LIN {X 0,Y 422.066,Z 378.159,A -85,B 0,C 180,E1 -10186.597,E2 -10186.597} C_VEL
LIN {X 0,Y 422.405,Z 363.356,A -85,B 0,C 180,E1 -10186.926,E2 -10186.926} C_VEL
LIN {X 0,Y 423.125,Z 289.794,A -85,B 0,C 180,E1 -10188.266,E2 -10188.266} C_VEL
LIN {X 0,Y 419.451,Z 264.662,A -85,B 0,C 180,E1 -10188.909,E2 -10188.909} C_VEL
LIN {X 0,Y 420.506,Z 247.774,A -85,B 0,C 180,E1 -10192.086,E2 -10192.086} C_VEL
LIN {X 0,Y 421.39,Z 234.372,A -85,B 0,C 180,E1 -10194.639,E2 -10194.639} C_VEL
LIN {X 0,Y 420.674,Z 228.931,A -85,B 0,C 180,E1 -10195.742,E2 -10195.742} C_VEL
LIN {X 0,Y 418.333,Z 217.378,A -85,B 0,C 180,E1 -10198.193,E2 -10198.193} C_VEL
LIN {X 0,Y 418.2,Z 217.392,A -85,B 0,C 180,E1 -10201.393,E2 -10201.393} C_VEL
LIN {X 0,Y 418.252,Z 217.383,A -85,B 0,C 180,E1 -10204.577,E2 -10204.577} C_VEL
LIN {X 0,Y 418.211,Z 217.393,A -85,B 0,C 180,E1 -10207.83,E2 -10207.83} C_VEL
LIN {X 0,Y 418.203,Z 217.388,A -85,B 0,C 180,E1 -10210.945,E2 -10210.945} C_VEL
LIN {X 0,Y 418.188,Z 217.396,A -85,B 0,C 180,E1 -10213.726,E2 -10213.726} C_VEL
LIN {X 0,Y 418.184,Z 217.391,A -85,B 0,C 180,E1 -10216.445,E2 -10216.445} C_VEL
LIN {X 0,Y 418.196,Z 217.39,A -85,B 0,C 180,E1 -10219.127,E2 -10219.127} C_VEL
LIN {X 0,Y 418.195,Z 217.391,A -85,B 0,C 180,E1 -10222.164,E2 -10222.164} C_VEL
LIN {X 0,Y 418.234,Z 217.389,A -85,B 0,C 180,E1 -10225.417,E2 -10225.417} C_VEL
LIN {X 0,Y 418.176,Z 217.391,A -85,B 0,C 180,E1 -10228.601,E2 -10228.601} C_VEL
LIN {X 0,Y 418.254,Z 217.384,A -85,B 0,C 180,E1 -10231.934,E2 -10231.934} C_VEL
LIN {X 0,Y 418.253,Z 217.386,A -85,B 0,C 180,E1 -10235.16,E2 -10235.16} C_VEL
LIN {X 0,Y 418.192,Z 217.389,A -85,B 0,C 180,E1 -10238.301,E2 -10238.301} C_VEL
LIN {X 0,Y 418.24,Z 217.389,A -85,B 0,C 180,E1 -10241.381,E2 -10241.381} C_VEL
LIN {X 0,Y 418.255,Z 217.381,A -85,B 0,C 180,E1 -10244.404,E2 -10244.404} C_VEL
LIN {X 0,Y 418.324,Z 217.377,A -85,B 0,C 180,E1 -10247.384,E2 -10247.384} C_VEL
LIN {X 0,Y 418.297,Z 217.376,A -85,B 0,C 180,E1 -10250.327,E2 -10250.327} C_VEL
LIN {X 0,Y 418.44,Z 217.363,A -85,B 0,C 180,E1 -10253.248,E2 -10253.248} C_VEL
LIN {X 0,Y 418.287,Z 217.383,A -85,B 0,C 180,E1 -10255.181,E2 -10255.181} C_VEL
LIN {X 0,Y 418.492,Z 217.352,A -85,B 0,C 180,E1 -10258.075,E2 -10258.075} C_VEL
LIN {X 0,Y 418.62,Z 217.336,A -85,B 0,C 180,E1 -10260,E2 -10260} C_VEL
LIN {X 0,Y 418.452,Z 217.364,A -85,B 0,C 180,E1 -10262.888,E2 -10262.888} C_VEL
LIN {X 0,Y 418.491,Z 217.352,A -85,B 0,C 180,E1 -10265.783,E2 -10265.783} C_VEL
LIN {X 0,Y 418.354,Z 217.376,A -85,B 0,C 180,E1 -10268.696,E2 -10268.696} C_VEL
LIN {X 0,Y 418.289,Z 217.377,A -85,B 0,C 180,E1 -10271.631,E2 -10271.631} C_VEL
LIN {X 0,Y 418.264,Z 217.387,A -85,B 0,C 180,E1 -10274.598,E2 -10274.598} C_VEL
LIN {X 0,Y 418.244,Z 217.383,A -85,B 0,C 180,E1 -10277.605,E2 -10277.605} C_VEL
LIN {X 0,Y 418.245,Z 217.388,A -85,B 0,C 180,E1 -10280.663,E2 -10280.663} C_VEL
LIN {X 0,Y 418.263,Z 217.381,A -85,B 0,C 180,E1 -10283.782,E2 -10283.782} C_VEL
LIN {X 0,Y 418.272,Z 217.38,A -85,B 0,C 180,E1 -10287.073,E2 -10287.073} C_VEL
LIN {X 0,Y 418.222,Z 217.392,A -85,B 0,C 180,E1 -10290.274,E2 -10290.274} C_VEL
LIN {X 0,Y 418.213,Z 217.388,A -85,B 0,C 180,E1 -10293.68,E2 -10293.68} C_VEL
LIN {X 0,Y 418.214,Z 217.386,A -85,B 0,C 180,E1 -10297.226,E2 -10297.226} C_VEL
LIN {X 0,Y 418.237,Z 217.385,A -85,B 0,C 180,E1 -10299.683,E2 -10299.683} C_VEL
LIN {X 0,Y 418.256,Z 217.386,A -85,B 0,C 180,E1 -10302.332,E2 -10302.332} C_VEL
LIN {X 0,Y 418.219,Z 217.386,A -85,B 0,C 180,E1 -10305.113,E2 -10305.113} C_VEL
LIN {X 0,Y 418.232,Z 217.388,A -85,B 0,C 180,E1 -10307.772,E2 -10307.772} C_VEL
LIN {X 0,Y 418.245,Z 217.383,A -85,B 0,C 180,E1 -10310.62,E2 -10310.62} C_VEL
LIN {X 0,Y 418.227,Z 217.391,A -85,B 0,C 180,E1 -10313.979,E2 -10313.979} C_VEL
LIN {X 0,Y 418.241,Z 217.384,A -85,B 0,C 180,E1 -10317.159,E2 -10317.159} C_VEL
LIN {X 0,Y 418.261,Z 217.381,A -85,B 0,C 180,E1 -10320.841,E2 -10320.841} C_VEL
LIN {X 0,Y 418.26,Z 217.383,A -85,B 0,C 180,E1 -10324.098,E2 -10324.098} C_VEL
LIN {X 0,Y 418.229,Z 217.387,A -85,B 0,C 180,E1 -10327.266,E2 -10327.266} C_VEL
LIN {X 0,Y 418.276,Z 217.379,A -85,B 0,C 180,E1 -10330.366,E2 -10330.366} C_VEL
LIN {X 0,Y 418.312,Z 217.38,A -85,B 0,C 180,E1 -10333.406,E2 -10333.406} C_VEL
LIN {X 0,Y 418.342,Z 217.373,A -85,B 0,C 180,E1 -10337.001,E2 -10337.001} C_VEL
LIN {X 0,Y 418.339,Z 217.371,A -85,B 0,C 180,E1 -10340.33,E2 -10340.33} C_VEL
LIN {X 0,Y 418.485,Z 217.359,A -85,B 0,C 180,E1 -10343.25,E2 -10343.25} C_VEL
LIN {X 0,Y 418.336,Z 217.377,A -85,B 0,C 180,E1 -10345.182,E2 -10345.182} C_VEL
LIN {X 0,Y 418.542,Z 217.346,A -85,B 0,C 180,E1 -10348.076,E2 -10348.076} C_VEL
LIN {X 0,Y 418.67,Z 217.33,A -85,B 0,C 180,E1 -10350,E2 -10350} C_VEL
LIN {X 0,Y 418.509,Z 217.354,A -85,B 0,C 180,E1 -10352.887,E2 -10352.887} C_VEL
LIN {X 0,Y 418.501,Z 217.351,A -85,B 0,C 180,E1 -10355.782,E2 -10355.782} C_VEL
LIN {X 0,Y 418.394,Z 217.367,A -85,B 0,C 180,E1 -10358.694,E2 -10358.694} C_VEL
LIN {X 0,Y 418.313,Z 217.375,A -85,B 0,C 180,E1 -10361.63,E2 -10361.63} C_VEL
LIN {X 0,Y 418.316,Z 217.376,A -85,B 0,C 180,E1 -10363.378,E2 -10363.378} C_VEL
LIN {X 0,Y 417.625,Z 217.461,A -85,B 0,C 180,E1 -10364.181,E2 -10364.181} C_VEL
LIN {X 0,Y 414.745,Z 217.82,A -85,B 0,C 180,E1 -10365.486,E2 -10365.486} C_VEL
LIN {X 0,Y 412.331,Z 218.122,A -85,B 0,C 180,E1 -10366.54,E2 -10366.54} C_VEL
LIN {X 0,Y 411.31,Z 218.249,A -85,B 0,C 180,E1 -10367.355,E2 -10367.355} C_VEL
LIN {X 0,Y 411.235,Z 218.256,A -85,B 0,C 180,E1 -10367.631,E2 -10367.631} C_VEL
LIN {X 0,Y 411.189,Z 218.266,A -85,B 0,C 180,E1 -10371.032,E2 -10371.032} C_VEL
LIN {X 0,Y 411.211,Z 218.26,A -85,B 0,C 180,E1 -10374.214,E2 -10374.214} C_VEL
LIN {X 0,Y 411.253,Z 218.258,A -85,B 0,C 180,E1 -10377.475,E2 -10377.475} C_VEL
LIN {X 0,Y 411.299,Z 218.345,A -85,B 0,C 180,E1 -10378.511,E2 -10378.511} C_VEL
LIN {X 0,Y 412.921,Z 227.389,A -85,B 0,C 180,E1 -10380.701,E2 -10380.701} C_VEL
LIN {X 0,Y 412.961,Z 228.338,A -85,B 0,C 180,E1 -10380.91,E2 -10380.91} C_VEL
LIN {X 0,Y 416.873,Z 248.303,A -85,B 0,C 180,E1 -10381.469,E2 -10381.469} C_VEL
LIN {X 0,Y 415.524,Z 335.93,A -85,B 0,C 180,E1 -10383.106,E2 -10383.106} C_VEL
LIN {X 0,Y 415.093,Z 349.118,A -85,B 0,C 180,E1 -10383.544,E2 -10383.544} C_VEL
LIN {X 0,Y 414.718,Z 361.357,A -85,B 0,C 180,E1 -10384.145,E2 -10384.145} C_VEL
LIN {X 0,Y 414.124,Z 373.394,A -85,B 0,C 180,E1 -10384.939,E2 -10384.939} C_VEL
LIN {X 0,Y 413.426,Z 384.953,A -85,B 0,C 180,E1 -10385.923,E2 -10385.923} C_VEL
LIN {X 0,Y 412.769,Z 395.514,A -85,B 0,C 180,E1 -10387.049,E2 -10387.049} C_VEL
LIN {X 0,Y 412.088,Z 405.097,A -85,B 0,C 180,E1 -10388.325,E2 -10388.325} C_VEL
LIN {X 0,Y 411.513,Z 413.918,A -85,B 0,C 180,E1 -10389.778,E2 -10389.778} C_VEL
LIN {X 0,Y 410.989,Z 420.898,A -85,B 0,C 180,E1 -10391.201,E2 -10391.201} C_VEL
LIN {X 0,Y 410.643,Z 426.469,A -85,B 0,C 180,E1 -10392.615,E2 -10392.615} C_VEL
LIN {X 0,Y 410.38,Z 430.837,A -85,B 0,C 180,E1 -10394.006,E2 -10394.006} C_VEL
LIN {X 0,Y 410.192,Z 434.163,A -85,B 0,C 180,E1 -10395.375,E2 -10395.375} C_VEL
LIN {X 0,Y 410.001,Z 436.573,A -85,B 0,C 180,E1 -10396.713,E2 -10396.713} C_VEL
LIN {X 0,Y 409.91,Z 438.196,A -85,B 0,C 180,E1 -10398.036,E2 -10398.036} C_VEL
LIN {X 0,Y 409.864,Z 439.072,A -85,B 0,C 180,E1 -10399.339,E2 -10399.339} C_VEL
LIN {X 0,Y 409.87,Z 439.206,A -85,B 0,C 180,E1 -10400.622,E2 -10400.622} C_VEL
LIN {X 0,Y 409.899,Z 438.569,A -85,B 0,C 180,E1 -10402.056,E2 -10402.056} C_VEL
LIN {X 0,Y 410.047,Z 436.829,A -85,B 0,C 180,E1 -10403.655,E2 -10403.655} C_VEL
LIN {X 0,Y 410.286,Z 433.278,A -85,B 0,C 180,E1 -10405.579,E2 -10405.579} C_VEL
LIN {X 0,Y 410.745,Z 427.943,A -85,B 0,C 180,E1 -10407.486,E2 -10407.486} C_VEL
LIN {X 0,Y 411.237,Z 421.689,A -85,B 0,C 180,E1 -10409.157,E2 -10409.157} C_VEL
LIN {X 0,Y 411.863,Z 414.212,A -85,B 0,C 180,E1 -10410.706,E2 -10410.706} C_VEL
LIN {X 0,Y 412.617,Z 405.207,A -85,B 0,C 180,E1 -10412.198,E2 -10412.198} C_VEL
LIN {X 0,Y 413.328,Z 395.464,A -85,B 0,C 180,E1 -10413.491,E2 -10413.491} C_VEL
LIN {X 0,Y 414.031,Z 385.541,A -85,B 0,C 180,E1 -10414.554,E2 -10414.554} C_VEL
LIN {X 0,Y 414.867,Z 374.104,A -85,B 0,C 180,E1 -10415.532,E2 -10415.532} C_VEL
LIN {X 0,Y 415.491,Z 362.385,A -85,B 0,C 180,E1 -10416.314,E2 -10416.314} C_VEL
LIN {X 0,Y 416.081,Z 349.135,A -85,B 0,C 180,E1 -10416.959,E2 -10416.959} C_VEL
LIN {X 0,Y 416.423,Z 336.373,A -85,B 0,C 180,E1 -10417.382,E2 -10417.382} C_VEL
LIN {X 0,Y 417.941,Z 247.923,A -85,B 0,C 180,E1 -10419.072,E2 -10419.072} C_VEL
LIN {X 0,Y 413.701,Z 229.623,A -85,B 0,C 180,E1 -10419.685,E2 -10419.685} C_VEL
LIN {X 0,Y 413.487,Z 228.755,A -85,B 0,C 180,E1 -10419.738,E2 -10419.738} C_VEL
LIN {X 0,Y 411.235,Z 218.26,A -85,B 0,C 180,E1 -10422.085,E2 -10422.085} C_VEL
LIN {X 0,Y 411.222,Z 218.266,A -85,B 0,C 180,E1 -10425.146,E2 -10425.146} C_VEL
LIN {X 0,Y 411.257,Z 218.262,A -85,B 0,C 180,E1 -10428.167,E2 -10428.167} C_VEL
LIN {X 0,Y 411.4,Z 218.239,A -85,B 0,C 180,E1 -10432.185,E2 -10432.185} C_VEL
LIN {X 0,Y 411.448,Z 218.232,A -85,B 0,C 180,E1 -10434.118,E2 -10434.118} C_VEL
LIN {X 0,Y 411.462,Z 218.23,A -85,B 0,C 180,E1 -10438.043,E2 -10438.043} C_VEL
LIN {X 0,Y 411.591,Z 218.214,A -85,B 0,C 180,E1 -10440,E2 -10440} C_VEL
LIN {X 0,Y 411.409,Z 218.239,A -85,B 0,C 180,E1 -10442.938,E2 -10442.938} C_VEL
LIN {X 0,Y 411.406,Z 218.24,A -85,B 0,C 180,E1 -10446.868,E2 -10446.868} C_VEL
LIN {X 0,Y 411.251,Z 218.255,A -85,B 0,C 180,E1 -10449.84,E2 -10449.84} C_VEL
LIN {X 0,Y 411.27,Z 218.255,A -85,B 0,C 180,E1 -10453.109,E2 -10453.109} C_VEL
LIN {X 0,Y 411.22,Z 218.259,A -85,B 0,C 180,E1 -10456.891,E2 -10456.891} C_VEL
LIN {X 0,Y 411.17,Z 218.265,A -85,B 0,C 180,E1 -10459.99,E2 -10459.99} C_VEL
LIN {X 0,Y 411.158,Z 218.264,A -85,B 0,C 180,E1 -10463.151,E2 -10463.151} C_VEL
LIN {X 0,Y 411.202,Z 218.263,A -85,B 0,C 180,E1 -10466.384,E2 -10466.384} C_VEL
LIN {X 0,Y 411.166,Z 218.262,A -85,B 0,C 180,E1 -10469.716,E2 -10469.716} C_VEL
LIN {X 0,Y 411.176,Z 218.264,A -85,B 0,C 180,E1 -10473.159,E2 -10473.159} C_VEL
LIN {X 0,Y 411.163,Z 218.271,A -85,B 0,C 180,E1 -10476.555,E2 -10476.555} C_VEL
LIN {X 0,Y 411.181,Z 218.266,A -85,B 0,C 180,E1 -10479.73,E2 -10479.73} C_VEL
LIN {X 0,Y 411.148,Z 218.265,A -85,B 0,C 180,E1 -10483.137,E2 -10483.137} C_VEL
LIN {X 0,Y 411.147,Z 218.269,A -85,B 0,C 180,E1 -10485.885,E2 -10485.885} C_VEL
LIN {X 0,Y 411.145,Z 218.27,A -85,B 0,C 180,E1 -10488.775,E2 -10488.775} C_VEL
LIN {X 0,Y 411.177,Z 218.268,A -85,B 0,C 180,E1 -10492.029,E2 -10492.029} C_VEL
LIN {X 0,Y 411.193,Z 218.266,A -85,B 0,C 180,E1 -10495.67,E2 -10495.67} C_VEL
LIN {X 0,Y 411.179,Z 218.267,A -85,B 0,C 180,E1 -10499.155,E2 -10499.155} C_VEL
LIN {X 0,Y 411.273,Z 218.415,A -85,B 0,C 180,E1 -10501.627,E2 -10501.627} C_VEL
LIN {X 0,Y 413.841,Z 230.347,A -85,B 0,C 180,E1 -10504.167,E2 -10504.167} C_VEL
LIN {X 0,Y 414.527,Z 235.409,A -85,B 0,C 180,E1 -10505.192,E2 -10505.192} C_VEL
LIN {X 0,Y 413.41,Z 251.975,A -85,B 0,C 180,E1 -10508.302,E2 -10508.302} C_VEL
LIN {X 0,Y 412.777,Z 262.59,A -85,B 0,C 180,E1 -10510.278,E2 -10510.278} C_VEL
LIN {X 0,Y 416.024,Z 282.027,A -85,B 0,C 180,E1 -10510.862,E2 -10510.862} C_VEL
LIN {X 0,Y 417.333,Z 292.66,A -85,B 0,C 180,E1 -10511.141,E2 -10511.141} C_VEL
LIN {X 0,Y 416.124,Z 372.966,A -85,B 0,C 180,E1 -10512.684,E2 -10512.684} C_VEL
LIN {X 0,Y 415.444,Z 386.355,A -85,B 0,C 180,E1 -10513.13,E2 -10513.13} C_VEL
LIN {X 0,Y 414.759,Z 399.136,A -85,B 0,C 180,E1 -10513.766,E2 -10513.766} C_VEL
LIN {X 0,Y 413.911,Z 411.684,A -85,B 0,C 180,E1 -10514.617,E2 -10514.617} C_VEL
LIN {X 0,Y 413.088,Z 423.323,A -85,B 0,C 180,E1 -10515.632,E2 -10515.632} C_VEL
LIN {X 0,Y 412.332,Z 433.101,A -85,B 0,C 180,E1 -10516.698,E2 -10516.698} C_VEL
LIN {X 0,Y 411.651,Z 442.324,A -85,B 0,C 180,E1 -10517.929,E2 -10517.929} C_VEL
LIN {X 0,Y 410.915,Z 451.346,A -85,B 0,C 180,E1 -10519.406,E2 -10519.406} C_VEL
LIN {X 0,Y 410.467,Z 458.597,A -85,B 0,C 180,E1 -10520.888,E2 -10520.888} C_VEL
LIN {X 0,Y 410.176,Z 465.224,A -85,B 0,C 180,E1 -10522.617,E2 -10522.617} C_VEL
LIN {X 0,Y 409.99,Z 469.606,A -85,B 0,C 180,E1 -10524.097,E2 -10524.097} C_VEL
LIN {X 0,Y 410.011,Z 471.94,A -85,B 0,C 180,E1 -10525.084,E2 -10525.084} C_VEL
LIN {X 0,Y 409.941,Z 473.79,A -85,B 0,C 180,E1 -10526.068,E2 -10526.068} C_VEL
LIN {X 0,Y 409.971,Z 475.198,A -85,B 0,C 180,E1 -10527.052,E2 -10527.052} C_VEL
LIN {X 0,Y 410.019,Z 476.203,A -85,B 0,C 180,E1 -10528.036,E2 -10528.036} C_VEL
LIN {X 0,Y 409.981,Z 476.805,A -85,B 0,C 180,E1 -10529.018,E2 -10529.018} C_VEL
LIN {X 0,Y 409.976,Z 476.961,A -85,B 0,C 180,E1 -10530,E2 -10530} C_VEL
LIN {X 0,Y 409.981,Z 476.707,A -85,B 0,C 180,E1 -10530.982,E2 -10530.982} C_VEL
LIN {X 0,Y 410.018,Z 476.057,A -85,B 0,C 180,E1 -10531.964,E2 -10531.964} C_VEL
LIN {X 0,Y 409.972,Z 474.998,A -85,B 0,C 180,E1 -10532.947,E2 -10532.947} C_VEL
LIN {X 0,Y 409.941,Z 473.471,A -85,B 0,C 180,E1 -10533.932,E2 -10533.932} C_VEL
LIN {X 0,Y 410.024,Z 470.372,A -85,B 0,C 180,E1 -10535.409,E2 -10535.409} C_VEL
LIN {X 0,Y 410.163,Z 466.182,A -85,B 0,C 180,E1 -10536.888,E2 -10536.888} C_VEL
LIN {X 0,Y 410.384,Z 459.759,A -85,B 0,C 180,E1 -10538.617,E2 -10538.617} C_VEL
LIN {X 0,Y 410.732,Z 452.748,A -85,B 0,C 180,E1 -10540.1,E2 -10540.1} C_VEL
LIN {X 0,Y 411.32,Z 443.951,A -85,B 0,C 180,E1 -10541.58,E2 -10541.58} C_VEL
LIN {X 0,Y 411.92,Z 434.928,A -85,B 0,C 180,E1 -10542.813,E2 -10542.813} C_VEL
LIN {X 0,Y 412.682,Z 424.044,A -85,B 0,C 180,E1 -10544.018,E2 -10544.018} C_VEL
LIN {X 0,Y 413.345,Z 412.491,A -85,B 0,C 180,E1 -10545.026,E2 -10545.026} C_VEL
LIN {X 0,Y 414.169,Z 399.868,A -85,B 0,C 180,E1 -10545.878,E2 -10545.878} C_VEL
LIN {X 0,Y 414.792,Z 387.64,A -85,B 0,C 180,E1 -10546.485,E2 -10546.485} C_VEL
LIN {X 0,Y 415.304,Z 374.278,A -85,B 0,C 180,E1 -10546.939,E2 -10546.939} C_VEL
LIN {X 0,Y 415.985,Z 331.19,A -85,B 0,C 180,E1 -10547.758,E2 -10547.758} C_VEL
LIN {X 0,Y 416.299,Z 290.521,A -85,B 0,C 180,E1 -10548.523,E2 -10548.523} C_VEL
LIN {X 0,Y 412.517,Z 264.36,A -85,B 0,C 180,E1 -10549.207,E2 -10549.207} C_VEL
LIN {X 0,Y 413.63,Z 247.327,A -85,B 0,C 180,E1 -10552.473,E2 -10552.473} C_VEL
LIN {X 0,Y 414.434,Z 235.243,A -85,B 0,C 180,E1 -10554.813,E2 -10554.813} C_VEL
LIN {X 0,Y 413.608,Z 229.802,A -85,B 0,C 180,E1 -10555.941,E2 -10555.941} C_VEL
LIN {X 0,Y 411.291,Z 218.254,A -85,B 0,C 180,E1 -10558.442,E2 -10558.442} C_VEL
LIN {X 0,Y 411.154,Z 218.273,A -85,B 0,C 180,E1 -10561.994,E2 -10561.994} C_VEL
LIN {X 0,Y 411.197,Z 218.261,A -85,B 0,C 180,E1 -10564.875,E2 -10564.875} C_VEL
LIN {X 0,Y 411.186,Z 218.266,A -85,B 0,C 180,E1 -10568.165,E2 -10568.165} C_VEL
LIN {X 0,Y 411.144,Z 218.268,A -85,B 0,C 180,E1 -10571.225,E2 -10571.225} C_VEL
LIN {X 0,Y 411.154,Z 218.267,A -85,B 0,C 180,E1 -10574.487,E2 -10574.487} C_VEL
LIN {X 0,Y 411.151,Z 218.268,A -85,B 0,C 180,E1 -10578.191,E2 -10578.191} C_VEL
LIN {X 0,Y 411.18,Z 218.263,A -85,B 0,C 180,E1 -10580.771,E2 -10580.771} C_VEL
LIN {X 0,Y 411.167,Z 218.264,A -85,B 0,C 180,E1 -10584.468,E2 -10584.468} C_VEL
LIN {X 0,Y 411.176,Z 218.264,A -85,B 0,C 180,E1 -10586.87,E2 -10586.87} C_VEL
LIN {X 0,Y 411.18,Z 218.263,A -85,B 0,C 180,E1 -10590.646,E2 -10590.646} C_VEL
LIN {X 0,Y 411.2,Z 218.265,A -85,B 0,C 180,E1 -10593.616,E2 -10593.616} C_VEL
LIN {X 0,Y 411.157,Z 218.267,A -85,B 0,C 180,E1 -10596.849,E2 -10596.849} C_VEL
LIN {X 0,Y 411.172,Z 218.264,A -85,B 0,C 180,E1 -10600.049,E2 -10600.049} C_VEL
LIN {X 0,Y 411.222,Z 218.263,A -85,B 0,C 180,E1 -10603.129,E2 -10603.129} C_VEL
LIN {X 0,Y 411.269,Z 218.255,A -85,B 0,C 180,E1 -10606.891,E2 -10606.891} C_VEL
LIN {X 0,Y 411.25,Z 218.254,A -85,B 0,C 180,E1 -10610.16,E2 -10610.16} C_VEL
LIN {X 0,Y 411.405,Z 218.241,A -85,B 0,C 180,E1 -10613.132,E2 -10613.132} C_VEL
LIN {X 0,Y 411.259,Z 218.259,A -85,B 0,C 180,E1 -10615.098,E2 -10615.098} C_VEL
LIN {X 0,Y 411.461,Z 218.228,A -85,B 0,C 180,E1 -10618.042,E2 -10618.042} C_VEL
LIN {X 0,Y 411.59,Z 218.212,A -85,B 0,C 180,E1 -10620,E2 -10620} C_VEL
LIN {X 0,Y 411.41,Z 218.241,A -85,B 0,C 180,E1 -10622.937,E2 -10622.937} C_VEL
LIN {X 0,Y 411.427,Z 218.237,A -85,B 0,C 180,E1 -10626.762,E2 -10626.762} C_VEL
LIN {X 0,Y 411.251,Z 218.254,A -85,B 0,C 180,E1 -10629.839,E2 -10629.839} C_VEL
LIN {X 0,Y 411.269,Z 218.254,A -85,B 0,C 180,E1 -10633.109,E2 -10633.109} C_VEL
LIN {X 0,Y 411.218,Z 218.262,A -85,B 0,C 180,E1 -10636.89,E2 -10636.89} C_VEL
LIN {X 0,Y 411.216,Z 218.26,A -85,B 0,C 180,E1 -10639.987,E2 -10639.987} C_VEL
LIN {X 0,Y 411.203,Z 218.261,A -85,B 0,C 180,E1 -10643.147,E2 -10643.147} C_VEL
LIN {X 0,Y 411.2,Z 218.267,A -85,B 0,C 180,E1 -10646.383,E2 -10646.383} C_VEL
LIN {X 0,Y 411.172,Z 218.264,A -85,B 0,C 180,E1 -10649.715,E2 -10649.715} C_VEL
LIN {X 0,Y 411.172,Z 218.264,A -85,B 0,C 180,E1 -10653.158,E2 -10653.158} C_VEL
LIN {X 0,Y 411.163,Z 218.268,A -85,B 0,C 180,E1 -10656.556,E2 -10656.556} C_VEL
LIN {X 0,Y 411.199,Z 218.263,A -85,B 0,C 180,E1 -10659.733,E2 -10659.733} C_VEL
LIN {X 0,Y 411.191,Z 218.261,A -85,B 0,C 180,E1 -10663.131,E2 -10663.131} C_VEL
LIN {X 0,Y 411.145,Z 218.272,A -85,B 0,C 180,E1 -10665.884,E2 -10665.884} C_VEL
LIN {X 0,Y 411.189,Z 218.263,A -85,B 0,C 180,E1 -10669.502,E2 -10669.502} C_VEL
LIN {X 0,Y 411.183,Z 218.268,A -85,B 0,C 180,E1 -10672.03,E2 -10672.03} C_VEL
LIN {X 0,Y 411.189,Z 218.266,A -85,B 0,C 180,E1 -10675.669,E2 -10675.669} C_VEL
LIN {X 0,Y 411.183,Z 218.263,A -85,B 0,C 180,E1 -10679.156,E2 -10679.156} C_VEL
LIN {X 0,Y 411.248,Z 218.254,A -85,B 0,C 180,E1 -10682.525,E2 -10682.525} C_VEL
LIN {X 0,Y 411.218,Z 218.264,A -85,B 0,C 180,E1 -10685.787,E2 -10685.787} C_VEL
LIN {X 0,Y 411.188,Z 218.263,A -85,B 0,C 180,E1 -10688.968,E2 -10688.968} C_VEL
LIN {X 0,Y 411.246,Z 218.256,A -85,B 0,C 180,E1 -10692.087,E2 -10692.087} C_VEL
LIN {X 0,Y 411.256,Z 218.256,A -85,B 0,C 180,E1 -10695.149,E2 -10695.149} C_VEL
LIN {X 0,Y 411.281,Z 218.251,A -85,B 0,C 180,E1 -10698.169,E2 -10698.169} C_VEL
LIN {X 0,Y 411.438,Z 218.231,A -85,B 0,C 180,E1 -10702.19,E2 -10702.19} C_VEL
LIN {X 0,Y 411.469,Z 218.227,A -85,B 0,C 180,E1 -10704.119,E2 -10704.119} C_VEL
LIN {X 0,Y 411.512,Z 218.222,A -85,B 0,C 180,E1 -10708.043,E2 -10708.043} C_VEL
LIN {X 0,Y 411.639,Z 218.206,A -85,B 0,C 180,E1 -10710,E2 -10710} C_VEL
LIN {X 0,Y 411.464,Z 218.232,A -85,B 0,C 180,E1 -10712.937,E2 -10712.937} C_VEL
LIN {X 0,Y 411.462,Z 218.228,A -85,B 0,C 180,E1 -10715.882,E2 -10715.882} C_VEL
LIN {X 0,Y 411.349,Z 218.246,A -85,B 0,C 180,E1 -10718.844,E2 -10718.844} C_VEL
LIN {X 0,Y 411.281,Z 218.25,A -85,B 0,C 180,E1 -10721.832,E2 -10721.832} C_VEL
LIN {X 0,Y 411.255,Z 218.26,A -85,B 0,C 180,E1 -10724.851,E2 -10724.851} C_VEL
LIN {X 0,Y 411.235,Z 218.256,A -85,B 0,C 180,E1 -10727.631,E2 -10727.631} C_VEL
LIN {X 0,Y 410.577,Z 218.342,A -85,B 0,C 180,E1 -10728.449,E2 -10728.449} C_VEL
LIN {X 0,Y 407.687,Z 218.698,A -85,B 0,C 180,E1 -10729.777,E2 -10729.777} C_VEL
LIN {X 0,Y 405.239,Z 219.009,A -85,B 0,C 180,E1 -10730.849,E2 -10730.849} C_VEL
LIN {X 0,Y 404.203,Z 219.132,A -85,B 0,C 180,E1 -10731.679,E2 -10731.679} C_VEL
LIN {X 0,Y 404.128,Z 219.141,A -85,B 0,C 180,E1 -10731.961,E2 -10731.961} C_VEL
LIN {X 0,Y 404.206,Z 219.136,A -85,B 0,C 180,E1 -10735.294,E2 -10735.294} C_VEL
LIN {X 0,Y 404.272,Z 219.247,A -85,B 0,C 180,E1 -10738.308,E2 -10738.308} C_VEL
LIN {X 0,Y 405.958,Z 228.546,A -85,B 0,C 180,E1 -10740.599,E2 -10740.599} C_VEL
LIN {X 0,Y 410.088,Z 248.762,A -85,B 0,C 180,E1 -10741.187,E2 -10741.187} C_VEL
LIN {X 0,Y 408.677,Z 336.018,A -85,B 0,C 180,E1 -10742.846,E2 -10742.846} C_VEL
LIN {X 0,Y 408.239,Z 349.273,A -85,B 0,C 180,E1 -10743.292,E2 -10743.292} C_VEL
LIN {X 0,Y 407.832,Z 361.592,A -85,B 0,C 180,E1 -10743.904,E2 -10743.904} C_VEL
LIN {X 0,Y 407.211,Z 373.686,A -85,B 0,C 180,E1 -10744.714,E2 -10744.714} C_VEL
LIN {X 0,Y 406.541,Z 384.676,A -85,B 0,C 180,E1 -10745.659,E2 -10745.659} C_VEL
LIN {X 0,Y 405.838,Z 395.27,A -85,B 0,C 180,E1 -10746.795,E2 -10746.795} C_VEL
LIN {X 0,Y 405.118,Z 405.412,A -85,B 0,C 180,E1 -10748.159,E2 -10748.159} C_VEL
LIN {X 0,Y 404.483,Z 414.468,A -85,B 0,C 180,E1 -10749.678,E2 -10749.678} C_VEL
LIN {X 0,Y 403.967,Z 421.065,A -85,B 0,C 180,E1 -10751.048,E2 -10751.048} C_VEL
LIN {X 0,Y 403.592,Z 426.547,A -85,B 0,C 180,E1 -10752.451,E2 -10752.451} C_VEL
LIN {X 0,Y 403.278,Z 431.818,A -85,B 0,C 180,E1 -10754.188,E2 -10754.188} C_VEL
LIN {X 0,Y 403.041,Z 435.368,A -85,B 0,C 180,E1 -10755.774,E2 -10755.774} C_VEL
LIN {X 0,Y 402.878,Z 437.538,A -85,B 0,C 180,E1 -10757.131,E2 -10757.131} C_VEL
LIN {X 0,Y 402.81,Z 439.001,A -85,B 0,C 180,E1 -10758.604,E2 -10758.604} C_VEL
LIN {X 0,Y 402.754,Z 439.581,A -85,B 0,C 180,E1 -10760.149,E2 -10760.149} C_VEL
LIN {X 0,Y 402.792,Z 439.176,A -85,B 0,C 180,E1 -10761.728,E2 -10761.728} C_VEL
LIN {X 0,Y 402.958,Z 437.329,A -85,B 0,C 180,E1 -10763.631,E2 -10763.631} C_VEL
LIN {X 0,Y 403.215,Z 433.917,A -85,B 0,C 180,E1 -10765.561,E2 -10765.561} C_VEL
LIN {X 0,Y 403.627,Z 429.286,A -85,B 0,C 180,E1 -10767.332,E2 -10767.332} C_VEL
LIN {X 0,Y 404.171,Z 422.865,A -85,B 0,C 180,E1 -10769.139,E2 -10769.139} C_VEL
LIN {X 0,Y 404.745,Z 416.268,A -85,B 0,C 180,E1 -10770.595,E2 -10770.595} C_VEL
LIN {X 0,Y 405.54,Z 407.726,A -85,B 0,C 180,E1 -10772.102,E2 -10772.102} C_VEL
LIN {X 0,Y 406.336,Z 398.021,A -85,B 0,C 180,E1 -10773.476,E2 -10773.476} C_VEL
LIN {X 0,Y 407.023,Z 388.568,A -85,B 0,C 180,E1 -10774.564,E2 -10774.564} C_VEL
LIN {X 0,Y 407.875,Z 377.625,A -85,B 0,C 180,E1 -10775.573,E2 -10775.573} C_VEL
LIN {X 0,Y 408.62,Z 365.339,A -85,B 0,C 180,E1 -10776.458,E2 -10776.458} C_VEL
LIN {X 0,Y 409.269,Z 352.687,A -85,B 0,C 180,E1 -10777.138,E2 -10777.138} C_VEL
LIN {X 0,Y 409.633,Z 339.747,A -85,B 0,C 180,E1 -10777.619,E2 -10777.619} C_VEL
LIN {X 0,Y 410.038,Z 318.579,A -85,B 0,C 180,E1 -10778.07,E2 -10778.07} C_VEL
LIN {X 0,Y 411.313,Z 248.954,A -85,B 0,C 180,E1 -10779.422,E2 -10779.422} C_VEL
LIN {X 0,Y 407.532,Z 232.418,A -85,B 0,C 180,E1 -10779.989,E2 -10779.989} C_VEL
LIN {X 0,Y 406.355,Z 229.099,A -85,B 0,C 180,E1 -10780.159,E2 -10780.159} C_VEL
LIN {X 0,Y 404.185,Z 219.138,A -85,B 0,C 180,E1 -10782.481,E2 -10782.481} C_VEL
LIN {X 0,Y 404.175,Z 219.145,A -85,B 0,C 180,E1 -10785.911,E2 -10785.911} C_VEL
LIN {X 0,Y 404.22,Z 219.14,A -85,B 0,C 180,E1 -10788.975,E2 -10788.975} C_VEL
LIN {X 0,Y 404.363,Z 219.116,A -85,B 0,C 180,E1 -10792.127,E2 -10792.127} C_VEL
LIN {X 0,Y 404.394,Z 219.111,A -85,B 0,C 180,E1 -10794.015,E2 -10794.015} C_VEL
LIN {X 0,Y 404.432,Z 219.106,A -85,B 0,C 180,E1 -10798.009,E2 -10798.009} C_VEL
LIN {X 0,Y 404.561,Z 219.09,A -85,B 0,C 180,E1 -10800,E2 -10800} C_VEL
LIN {X 0,Y 404.367,Z 219.116,A -85,B 0,C 180,E1 -10802.989,E2 -10802.989} C_VEL
LIN {X 0,Y 404.37,Z 219.11,A -85,B 0,C 180,E1 -10805.986,E2 -10805.986} C_VEL
LIN {X 0,Y 404.247,Z 219.13,A -85,B 0,C 180,E1 -10809.002,E2 -10809.002} C_VEL
LIN {X 0,Y 404.225,Z 219.129,A -85,B 0,C 180,E1 -10812.043,E2 -10812.043} C_VEL
LIN {X 0,Y 404.167,Z 219.141,A -85,B 0,C 180,E1 -10815.12,E2 -10815.12} C_VEL
LIN {X 0,Y 404.169,Z 219.137,A -85,B 0,C 180,E1 -10818.24,E2 -10818.24} C_VEL
LIN {X 0,Y 404.098,Z 219.147,A -85,B 0,C 180,E1 -10821.422,E2 -10821.422} C_VEL
LIN {X 0,Y 404.138,Z 219.145,A -85,B 0,C 180,E1 -10824.669,E2 -10824.669} C_VEL
LIN {X 0,Y 404.16,Z 219.139,A -85,B 0,C 180,E1 -10828.003,E2 -10828.003} C_VEL
LIN {X 0,Y 404.106,Z 219.145,A -85,B 0,C 180,E1 -10831.56,E2 -10831.56} C_VEL
LIN {X 0,Y 404.154,Z 219.137,A -85,B 0,C 180,E1 -10835.02,E2 -10835.02} C_VEL
LIN {X 0,Y 404.121,Z 219.147,A -85,B 0,C 180,E1 -10838.761,E2 -10838.761} C_VEL
LIN {X 0,Y 404.096,Z 219.147,A -85,B 0,C 180,E1 -10841.602,E2 -10841.602} C_VEL
LIN {X 0,Y 404.123,Z 219.145,A -85,B 0,C 180,E1 -10844.525,E2 -10844.525} C_VEL
LIN {X 0,Y 404.116,Z 219.144,A -85,B 0,C 180,E1 -10847.299,E2 -10847.299} C_VEL
LIN {X 0,Y 404.153,Z 219.142,A -85,B 0,C 180,E1 -10849.959,E2 -10849.959} C_VEL
LIN {X 0,Y 404.121,Z 219.145,A -85,B 0,C 180,E1 -10853.129,E2 -10853.129} C_VEL
LIN {X 0,Y 404.133,Z 219.146,A -85,B 0,C 180,E1 -10856.191,E2 -10856.191} C_VEL
LIN {X 0,Y 404.136,Z 219.147,A -85,B 0,C 180,E1 -10859.718,E2 -10859.718} C_VEL
LIN {X 0,Y 404.206,Z 219.204,A -85,B 0,C 180,E1 -10861.262,E2 -10861.262} C_VEL
LIN {X 0,Y 406.875,Z 231.415,A -85,B 0,C 180,E1 -10863.923,E2 -10863.923} C_VEL
LIN {X 0,Y 407.635,Z 236.681,A -85,B 0,C 180,E1 -10865.017,E2 -10865.017} C_VEL
LIN {X 0,Y 406.675,Z 250.473,A -85,B 0,C 180,E1 -10867.657,E2 -10867.657} C_VEL
LIN {X 0,Y 405.923,Z 262.373,A -85,B 0,C 180,E1 -10869.893,E2 -10869.893} C_VEL
LIN {X 0,Y 409.282,Z 281.914,A -85,B 0,C 180,E1 -10870.491,E2 -10870.491} C_VEL
LIN {X 0,Y 410.689,Z 294.318,A -85,B 0,C 180,E1 -10870.825,E2 -10870.825} C_VEL
LIN {X 0,Y 409.434,Z 372.565,A -85,B 0,C 180,E1 -10872.36,E2 -10872.36} C_VEL
LIN {X 0,Y 408.679,Z 386.7,A -85,B 0,C 180,E1 -10872.842,E2 -10872.842} C_VEL
LIN {X 0,Y 407.962,Z 399.241,A -85,B 0,C 180,E1 -10873.488,E2 -10873.488} C_VEL
LIN {X 0,Y 407.05,Z 411.699,A -85,B 0,C 180,E1 -10874.351,E2 -10874.351} C_VEL
LIN {X 0,Y 406.21,Z 422.891,A -85,B 0,C 180,E1 -10875.345,E2 -10875.345} C_VEL
LIN {X 0,Y 405.383,Z 433.348,A -85,B 0,C 180,E1 -10876.513,E2 -10876.513} C_VEL
LIN {X 0,Y 404.693,Z 442.162,A -85,B 0,C 180,E1 -10877.719,E2 -10877.719} C_VEL
LIN {X 0,Y 403.903,Z 451.142,A -85,B 0,C 180,E1 -10879.22,E2 -10879.22} C_VEL
LIN {X 0,Y 403.433,Z 458.35,A -85,B 0,C 180,E1 -10880.728,E2 -10880.728} C_VEL
LIN {X 0,Y 403.106,Z 464.961,A -85,B 0,C 180,E1 -10882.487,E2 -10882.487} C_VEL
LIN {X 0,Y 402.919,Z 469.331,A -85,B 0,C 180,E1 -10883.993,E2 -10883.993} C_VEL
LIN {X 0,Y 402.919,Z 471.658,A -85,B 0,C 180,E1 -10884.997,E2 -10884.997} C_VEL
LIN {X 0,Y 402.86,Z 473.493,A -85,B 0,C 180,E1 -10885.999,E2 -10885.999} C_VEL
LIN {X 0,Y 402.947,Z 475.895,A -85,B 0,C 180,E1 -10888.001,E2 -10888.001} C_VEL
LIN {X 0,Y 402.906,Z 476.485,A -85,B 0,C 180,E1 -10889.001,E2 -10889.001} C_VEL
LIN {X 0,Y 402.899,Z 476.627,A -85,B 0,C 180,E1 -10890,E2 -10890} C_VEL
LIN {X 0,Y 402.905,Z 476.364,A -85,B 0,C 180,E1 -10890.999,E2 -10890.999} C_VEL
LIN {X 0,Y 402.946,Z 475.705,A -85,B 0,C 180,E1 -10891.999,E2 -10891.999} C_VEL
LIN {X 0,Y 402.873,Z 474.628,A -85,B 0,C 180,E1 -10892.999,E2 -10892.999} C_VEL
LIN {X 0,Y 402.862,Z 473.085,A -85,B 0,C 180,E1 -10894.001,E2 -10894.001} C_VEL
LIN {X 0,Y 402.921,Z 469.959,A -85,B 0,C 180,E1 -10895.504,E2 -10895.504} C_VEL
LIN {X 0,Y 403.074,Z 465.742,A -85,B 0,C 180,E1 -10897.01,E2 -10897.01} C_VEL
LIN {X 0,Y 403.335,Z 459.287,A -85,B 0,C 180,E1 -10898.769,E2 -10898.769} C_VEL
LIN {X 0,Y 403.685,Z 452.233,A -85,B 0,C 180,E1 -10900.278,E2 -10900.278} C_VEL
LIN {X 0,Y 404.326,Z 443.381,A -85,B 0,C 180,E1 -10901.784,E2 -10901.784} C_VEL
LIN {X 0,Y 404.977,Z 434.306,A -85,B 0,C 180,E1 -10903.037,E2 -10903.037} C_VEL
LIN {X 0,Y 405.689,Z 424.33,A -85,B 0,C 180,E1 -10904.162,E2 -10904.162} C_VEL
LIN {X 0,Y 406.344,Z 413.266,A -85,B 0,C 180,E1 -10905.163,E2 -10905.163} C_VEL
LIN {X 0,Y 407.165,Z 400.918,A -85,B 0,C 180,E1 -10906.03,E2 -10906.03} C_VEL
LIN {X 0,Y 407.831,Z 389.291,A -85,B 0,C 180,E1 -10906.646,E2 -10906.646} C_VEL
LIN {X 0,Y 408.352,Z 377.028,A -85,B 0,C 180,E1 -10907.107,E2 -10907.107} C_VEL
LIN {X 0,Y 408.75,Z 360.306,A -85,B 0,C 180,E1 -10907.477,E2 -10907.477} C_VEL
LIN {X 0,Y 409.571,Z 291.834,A -85,B 0,C 180,E1 -10908.773,E2 -10908.773} C_VEL
LIN {X 0,Y 405.571,Z 264.062,A -85,B 0,C 180,E1 -10909.517,E2 -10909.517} C_VEL
LIN {X 0,Y 406.759,Z 246.836,A -85,B 0,C 180,E1 -10912.874,E2 -10912.874} C_VEL
LIN {X 0,Y 407.471,Z 236.105,A -85,B 0,C 180,E1 -10914.994,E2 -10914.994} C_VEL
LIN {X 0,Y 406.031,Z 227.898,A -85,B 0,C 180,E1 -10916.743,E2 -10916.743} C_VEL
LIN {X 0,Y 404.244,Z 219.132,A -85,B 0,C 180,E1 -10918.7,E2 -10918.7} C_VEL
LIN {X 0,Y 404.129,Z 219.144,A -85,B 0,C 180,E1 -10922.619,E2 -10922.619} C_VEL
LIN {X 0,Y 404.167,Z 219.137,A -85,B 0,C 180,E1 -10925.186,E2 -10925.186} C_VEL
LIN {X 0,Y 404.136,Z 219.14,A -85,B 0,C 180,E1 -10928.754,E2 -10928.754} C_VEL
LIN {X 0,Y 404.103,Z 219.148,A -85,B 0,C 180,E1 -10931.596,E2 -10931.596} C_VEL
LIN {X 0,Y 404.123,Z 219.142,A -85,B 0,C 180,E1 -10934.518,E2 -10934.518} C_VEL
LIN {X 0,Y 404.111,Z 219.145,A -85,B 0,C 180,E1 -10937.292,E2 -10937.292} C_VEL
LIN {X 0,Y 404.129,Z 219.145,A -85,B 0,C 180,E1 -10939.95,E2 -10939.95} C_VEL
LIN {X 0,Y 404.106,Z 219.146,A -85,B 0,C 180,E1 -10943.122,E2 -10943.122} C_VEL
LIN {X 0,Y 404.114,Z 219.144,A -85,B 0,C 180,E1 -10946.184,E2 -10946.184} C_VEL
LIN {X 0,Y 404.111,Z 219.148,A -85,B 0,C 180,E1 -10949.712,E2 -10949.712} C_VEL
LIN {X 0,Y 404.159,Z 219.141,A -85,B 0,C 180,E1 -10953.12,E2 -10953.12} C_VEL
LIN {X 0,Y 404.137,Z 219.146,A -85,B 0,C 180,E1 -10955.331,E2 -10955.331} C_VEL
LIN {X 0,Y 404.097,Z 219.145,A -85,B 0,C 180,E1 -10958.578,E2 -10958.578} C_VEL
LIN {X 0,Y 404.167,Z 219.138,A -85,B 0,C 180,E1 -10961.76,E2 -10961.76} C_VEL
LIN {X 0,Y 404.161,Z 219.14,A -85,B 0,C 180,E1 -10964.88,E2 -10964.88} C_VEL
LIN {X 0,Y 404.224,Z 219.129,A -85,B 0,C 180,E1 -10967.957,E2 -10967.957} C_VEL
LIN {X 0,Y 404.357,Z 219.113,A -85,B 0,C 180,E1 -10972.132,E2 -10972.132} C_VEL
LIN {X 0,Y 404.369,Z 219.111,A -85,B 0,C 180,E1 -10974.014,E2 -10974.014} C_VEL
LIN {X 0,Y 404.43,Z 219.103,A -85,B 0,C 180,E1 -10978.008,E2 -10978.008} C_VEL
LIN {X 0,Y 404.56,Z 219.087,A -85,B 0,C 180,E1 -10980,E2 -10980} C_VEL
LIN {X 0,Y 404.368,Z 219.117,A -85,B 0,C 180,E1 -10982.988,E2 -10982.988} C_VEL
LIN {X 0,Y 404.369,Z 219.114,A -85,B 0,C 180,E1 -10986.764,E2 -10986.764} C_VEL
LIN {X 0,Y 404.217,Z 219.13,A -85,B 0,C 180,E1 -10990.012,E2 -10990.012} C_VEL
LIN {X 0,Y 404.223,Z 219.131,A -85,B 0,C 180,E1 -10993.212,E2 -10993.212} C_VEL
LIN {X 0,Y 404.175,Z 219.138,A -85,B 0,C 180,E1 -10997.009,E2 -10997.009} C_VEL
LIN {X 0,Y 404.17,Z 219.141,A -85,B 0,C 180,E1 -11000.351,E2 -11000.351} C_VEL
LIN {X 0,Y 404.153,Z 219.138,A -85,B 0,C 180,E1 -11003.575,E2 -11003.575} C_VEL
LIN {X 0,Y 404.158,Z 219.139,A -85,B 0,C 180,E1 -11006.879,E2 -11006.879} C_VEL
LIN {X 0,Y 404.116,Z 219.149,A -85,B 0,C 180,E1 -11010.287,E2 -11010.287} C_VEL
LIN {X 0,Y 404.111,Z 219.145,A -85,B 0,C 180,E1 -11013.815,E2 -11013.815} C_VEL
LIN {X 0,Y 404.108,Z 219.144,A -85,B 0,C 180,E1 -11016.878,E2 -11016.878} C_VEL
LIN {X 0,Y 404.139,Z 219.146,A -85,B 0,C 180,E1 -11020.086,E2 -11020.086} C_VEL
LIN {X 0,Y 404.167,Z 219.136,A -85,B 0,C 180,E1 -11023.093,E2 -11023.093} C_VEL
LIN {X 0,Y 404.125,Z 219.147,A -85,B 0,C 180,E1 -11025.929,E2 -11025.929} C_VEL
LIN {X 0,Y 404.128,Z 219.142,A -85,B 0,C 180,E1 -11028.642,E2 -11028.642} C_VEL
LIN {X 0,Y 404.14,Z 219.142,A -85,B 0,C 180,E1 -11031.494,E2 -11031.494} C_VEL
LIN {X 0,Y 404.167,Z 219.136,A -85,B 0,C 180,E1 -11034.987,E2 -11034.987} C_VEL
LIN {X 0,Y 404.13,Z 219.141,A -85,B 0,C 180,E1 -11038.557,E2 -11038.557} C_VEL
LIN {X 0,Y 404.186,Z 219.138,A -85,B 0,C 180,E1 -11042.003,E2 -11042.003} C_VEL
LIN {X 0,Y 404.168,Z 219.139,A -85,B 0,C 180,E1 -11045.337,E2 -11045.337} C_VEL
LIN {X 0,Y 404.13,Z 219.141,A -85,B 0,C 180,E1 -11048.583,E2 -11048.583} C_VEL
LIN {X 0,Y 404.204,Z 219.136,A -85,B 0,C 180,E1 -11051.764,E2 -11051.764} C_VEL
LIN {X 0,Y 404.202,Z 219.133,A -85,B 0,C 180,E1 -11054.884,E2 -11054.884} C_VEL
LIN {X 0,Y 404.253,Z 219.127,A -85,B 0,C 180,E1 -11057.96,E2 -11057.96} C_VEL
LIN {X 0,Y 404.402,Z 219.107,A -85,B 0,C 180,E1 -11062.13,E2 -11062.13} C_VEL
LIN {X 0,Y 404.417,Z 219.106,A -85,B 0,C 180,E1 -11064.016,E2 -11064.016} C_VEL
LIN {X 0,Y 404.481,Z 219.098,A -85,B 0,C 180,E1 -11068.009,E2 -11068.009} C_VEL
LIN {X 0,Y 404.608,Z 219.082,A -85,B 0,C 180,E1 -11070,E2 -11070} C_VEL
LIN {X 0,Y 404.421,Z 219.11,A -85,B 0,C 180,E1 -11072.988,E2 -11072.988} C_VEL
LIN {X 0,Y 404.409,Z 219.106,A -85,B 0,C 180,E1 -11075.985,E2 -11075.985} C_VEL
LIN {X 0,Y 404.287,Z 219.128,A -85,B 0,C 180,E1 -11079,E2 -11079} C_VEL
LIN {X 0,Y 404.253,Z 219.126,A -85,B 0,C 180,E1 -11082.04,E2 -11082.04} C_VEL
LIN {X 0,Y 404.201,Z 219.137,A -85,B 0,C 180,E1 -11085.117,E2 -11085.117} C_VEL
LIN {X 0,Y 404.205,Z 219.133,A -85,B 0,C 180,E1 -11088.236,E2 -11088.236} C_VEL
LIN {X 0,Y 404.131,Z 219.142,A -85,B 0,C 180,E1 -11091.417,E2 -11091.417} C_VEL
LIN {X 0,Y 404.128,Z 219.141,A -85,B 0,C 180,E1 -11091.961,E2 -11091.961} C_VEL
LIN {X 0,Y 403.487,Z 219.228,A -85,B 0,C 180,E1 -11092.792,E2 -11092.792} C_VEL
LIN {X 0,Y 400.653,Z 219.583,A -85,B 0,C 180,E1 -11094.144,E2 -11094.144} C_VEL
LIN {X 0,Y 398.242,Z 219.883,A -85,B 0,C 180,E1 -11095.236,E2 -11095.236} C_VEL
LIN {X 0,Y 397.207,Z 220.009,A -85,B 0,C 180,E1 -11096.081,E2 -11096.081} C_VEL
LIN {X 0,Y 397.124,Z 220.018,A -85,B 0,C 180,E1 -11096.366,E2 -11096.366} C_VEL
LIN {X 0,Y 397.233,Z 220.153,A -85,B 0,C 180,E1 -11098.103,E2 -11098.103} C_VEL
LIN {X 0,Y 398.899,Z 228.83,A -85,B 0,C 180,E1 -11100.283,E2 -11100.283} C_VEL
LIN {X 0,Y 402.157,Z 243.843,A -85,B 0,C 180,E1 -11100.738,E2 -11100.738} C_VEL
LIN {X 0,Y 403.322,Z 249.919,A -85,B 0,C 180,E1 -11100.912,E2 -11100.912} C_VEL
LIN {X 0,Y 401.828,Z 336.887,A -85,B 0,C 180,E1 -11102.606,E2 -11102.606} C_VEL
LIN {X 0,Y 401.361,Z 350.395,A -85,B 0,C 180,E1 -11103.078,E2 -11103.078} C_VEL
LIN {X 0,Y 400.908,Z 363.147,A -85,B 0,C 180,E1 -11103.74,E2 -11103.74} C_VEL
LIN {X 0,Y 400.279,Z 375.048,A -85,B 0,C 180,E1 -11104.574,E2 -11104.574} C_VEL
LIN {X 0,Y 399.531,Z 386.418,A -85,B 0,C 180,E1 -11105.589,E2 -11105.589} C_VEL
LIN {X 0,Y 398.782,Z 397.215,A -85,B 0,C 180,E1 -11106.808,E2 -11106.808} C_VEL
LIN {X 0,Y 397.999,Z 406.894,A -85,B 0,C 180,E1 -11108.168,E2 -11108.168} C_VEL
LIN {X 0,Y 397.454,Z 414.774,A -85,B 0,C 180,E1 -11109.531,E2 -11109.531} C_VEL
LIN {X 0,Y 396.917,Z 421.377,A -85,B 0,C 180,E1 -11110.925,E2 -11110.925} C_VEL
LIN {X 0,Y 396.537,Z 426.79,A -85,B 0,C 180,E1 -11112.331,E2 -11112.331} C_VEL
LIN {X 0,Y 396.27,Z 431.186,A -85,B 0,C 180,E1 -11113.757,E2 -11113.757} C_VEL
LIN {X 0,Y 396.057,Z 434.672,A -85,B 0,C 180,E1 -11115.212,E2 -11115.212} C_VEL
LIN {X 0,Y 395.828,Z 437.296,A -85,B 0,C 180,E1 -11116.709,E2 -11116.709} C_VEL
LIN {X 0,Y 395.738,Z 439.014,A -85,B 0,C 180,E1 -11118.228,E2 -11118.228} C_VEL
LIN {X 0,Y 395.663,Z 439.921,A -85,B 0,C 180,E1 -11120.249,E2 -11120.249} C_VEL
LIN {X 0,Y 395.719,Z 439.609,A -85,B 0,C 180,E1 -11121.567,E2 -11121.567} C_VEL
LIN {X 0,Y 395.799,Z 438.496,A -85,B 0,C 180,E1 -11123.03,E2 -11123.03} C_VEL
LIN {X 0,Y 396.021,Z 436.159,A -85,B 0,C 180,E1 -11124.711,E2 -11124.711} C_VEL
LIN {X 0,Y 396.386,Z 431.982,A -85,B 0,C 180,E1 -11126.658,E2 -11126.658} C_VEL
LIN {X 0,Y 396.843,Z 427.356,A -85,B 0,C 180,E1 -11128.209,E2 -11128.209} C_VEL
LIN {X 0,Y 397.305,Z 422.035,A -85,B 0,C 180,E1 -11129.625,E2 -11129.625} C_VEL
LIN {X 0,Y 398.012,Z 414.418,A -85,B 0,C 180,E1 -11131.238,E2 -11131.238} C_VEL
LIN {X 0,Y 398.871,Z 405.585,A -85,B 0,C 180,E1 -11132.735,E2 -11132.735} C_VEL
LIN {X 0,Y 399.632,Z 395.856,A -85,B 0,C 180,E1 -11134.059,E2 -11134.059} C_VEL
LIN {X 0,Y 400.593,Z 384.691,A -85,B 0,C 180,E1 -11135.269,E2 -11135.269} C_VEL
LIN {X 0,Y 401.433,Z 373.188,A -85,B 0,C 180,E1 -11136.255,E2 -11136.255} C_VEL
LIN {X 0,Y 402.172,Z 361.082,A -85,B 0,C 180,E1 -11137.051,E2 -11137.051} C_VEL
LIN {X 0,Y 402.766,Z 347.994,A -85,B 0,C 180,E1 -11137.685,E2 -11137.685} C_VEL
LIN {X 0,Y 403.152,Z 335.665,A -85,B 0,C 180,E1 -11138.077,E2 -11138.077} C_VEL
LIN {X 0,Y 404.666,Z 249.644,A -85,B 0,C 180,E1 -11139.795,E2 -11139.795} C_VEL
LIN {X 0,Y 401.253,Z 234.733,A -85,B 0,C 180,E1 -11140.325,E2 -11140.325} C_VEL
LIN {X 0,Y 399.259,Z 229.493,A -85,B 0,C 180,E1 -11140.595,E2 -11140.595} C_VEL
LIN {X 0,Y 397.19,Z 220.011,A -85,B 0,C 180,E1 -11142.821,E2 -11142.821} C_VEL
LIN {X 0,Y 397.188,Z 220.015,A -85,B 0,C 180,E1 -11146.702,E2 -11146.702} C_VEL
LIN {X 0,Y 397.179,Z 220.014,A -85,B 0,C 180,E1 -11149.808,E2 -11149.808} C_VEL
LIN {X 0,Y 397.315,Z 219.997,A -85,B 0,C 180,E1 -11152.888,E2 -11152.888} C_VEL
LIN {X 0,Y 397.215,Z 220.007,A -85,B 0,C 180,E1 -11154.925,E2 -11154.925} C_VEL
LIN {X 0,Y 397.401,Z 219.982,A -85,B 0,C 180,E1 -11157.973,E2 -11157.973} C_VEL
LIN {X 0,Y 397.531,Z 219.966,A -85,B 0,C 180,E1 -11160,E2 -11160} C_VEL
LIN {X 0,Y 397.327,Z 219.992,A -85,B 0,C 180,E1 -11163.042,E2 -11163.042} C_VEL
LIN {X 0,Y 397.322,Z 219.988,A -85,B 0,C 180,E1 -11166.093,E2 -11166.093} C_VEL
LIN {X 0,Y 397.21,Z 220.007,A -85,B 0,C 180,E1 -11169.163,E2 -11169.163} C_VEL
LIN {X 0,Y 397.186,Z 220.007,A -85,B 0,C 180,E1 -11172.26,E2 -11172.26} C_VEL
LIN {X 0,Y 397.14,Z 220.014,A -85,B 0,C 180,E1 -11175.394,E2 -11175.394} C_VEL
LIN {X 0,Y 397.121,Z 220.018,A -85,B 0,C 180,E1 -11178.576,E2 -11178.576} C_VEL
LIN {X 0,Y 397.056,Z 220.024,A -85,B 0,C 180,E1 -11181.821,E2 -11181.821} C_VEL
LIN {X 0,Y 397.117,Z 220.016,A -85,B 0,C 180,E1 -11185.515,E2 -11185.515} C_VEL
LIN {X 0,Y 397.082,Z 220.023,A -85,B 0,C 180,E1 -11188.547,E2 -11188.547} C_VEL
LIN {X 0,Y 397.046,Z 220.027,A -85,B 0,C 180,E1 -11192.075,E2 -11192.075} C_VEL
LIN {X 0,Y 397.09,Z 220.016,A -85,B 0,C 180,E1 -11195.506,E2 -11195.506} C_VEL
LIN {X 0,Y 397.098,Z 220.021,A -85,B 0,C 180,E1 -11198.863,E2 -11198.863} C_VEL
LIN {X 0,Y 397.043,Z 220.029,A -85,B 0,C 180,E1 -11202.271,E2 -11202.271} C_VEL
LIN {X 0,Y 397.065,Z 220.021,A -85,B 0,C 180,E1 -11205.073,E2 -11205.073} C_VEL
LIN {X 0,Y 397.046,Z 220.026,A -85,B 0,C 180,E1 -11208.025,E2 -11208.025} C_VEL
LIN {X 0,Y 397.112,Z 220.018,A -85,B 0,C 180,E1 -11211.142,E2 -11211.142} C_VEL
LIN {X 0,Y 397.106,Z 220.02,A -85,B 0,C 180,E1 -11214.5,E2 -11214.5} C_VEL
LIN {X 0,Y 397.067,Z 220.026,A -85,B 0,C 180,E1 -11217.931,E2 -11217.931} C_VEL
LIN {X 0,Y 397.144,Z 220.055,A -85,B 0,C 180,E1 -11220.883,E2 -11220.883} C_VEL
LIN {X 0,Y 399.596,Z 230.868,A -85,B 0,C 180,E1 -11223.313,E2 -11223.313} C_VEL
LIN {X 0,Y 400.765,Z 237.999,A -85,B 0,C 180,E1 -11224.836,E2 -11224.836} C_VEL
LIN {X 0,Y 399.667,Z 253.143,A -85,B 0,C 180,E1 -11227.788,E2 -11227.788} C_VEL
LIN {X 0,Y 399.068,Z 261.834,A -85,B 0,C 180,E1 -11229.464,E2 -11229.464} C_VEL
LIN {X 0,Y 402.611,Z 282.35,A -85,B 0,C 180,E1 -11230.121,E2 -11230.121} C_VEL
LIN {X 0,Y 404.082,Z 293.773,A -85,B 0,C 180,E1 -11230.445,E2 -11230.445} C_VEL
LIN {X 0,Y 402.721,Z 372.277,A -85,B 0,C 180,E1 -11232.023,E2 -11232.023} C_VEL
LIN {X 0,Y 401.956,Z 386.336,A -85,B 0,C 180,E1 -11232.513,E2 -11232.513} C_VEL
LIN {X 0,Y 401.172,Z 399.347,A -85,B 0,C 180,E1 -11233.2,E2 -11233.2} C_VEL
LIN {X 0,Y 400.219,Z 411.715,A -85,B 0,C 180,E1 -11234.077,E2 -11234.077} C_VEL
LIN {X 0,Y 399.332,Z 422.828,A -85,B 0,C 180,E1 -11235.086,E2 -11235.086} C_VEL
LIN {X 0,Y 398.432,Z 433.614,A -85,B 0,C 180,E1 -11236.323,E2 -11236.323} C_VEL
LIN {X 0,Y 397.581,Z 443.673,A -85,B 0,C 180,E1 -11237.755,E2 -11237.755} C_VEL
LIN {X 0,Y 396.794,Z 452.251,A -85,B 0,C 180,E1 -11239.283,E2 -11239.283} C_VEL
LIN {X 0,Y 396.324,Z 459.173,A -85,B 0,C 180,E1 -11240.817,E2 -11240.817} C_VEL
LIN {X 0,Y 396.04,Z 464.721,A -85,B 0,C 180,E1 -11242.352,E2 -11242.352} C_VEL
LIN {X 0,Y 395.842,Z 469.066,A -85,B 0,C 180,E1 -11243.885,E2 -11243.885} C_VEL
LIN {X 0,Y 395.828,Z 471.381,A -85,B 0,C 180,E1 -11244.907,E2 -11244.907} C_VEL
LIN {X 0,Y 395.781,Z 473.2,A -85,B 0,C 180,E1 -11245.927,E2 -11245.927} C_VEL
LIN {X 0,Y 395.857,Z 475.586,A -85,B 0,C 180,E1 -11247.965,E2 -11247.965} C_VEL
LIN {X 0,Y 395.833,Z 476.164,A -85,B 0,C 180,E1 -11248.983,E2 -11248.983} C_VEL
LIN {X 0,Y 395.823,Z 476.293,A -85,B 0,C 180,E1 -11250,E2 -11250} C_VEL
LIN {X 0,Y 395.833,Z 476.021,A -85,B 0,C 180,E1 -11251.017,E2 -11251.017} C_VEL
LIN {X 0,Y 395.875,Z 475.353,A -85,B 0,C 180,E1 -11252.034,E2 -11252.034} C_VEL
LIN {X 0,Y 395.775,Z 474.257,A -85,B 0,C 180,E1 -11253.053,E2 -11253.053} C_VEL
LIN {X 0,Y 395.785,Z 472.7,A -85,B 0,C 180,E1 -11254.073,E2 -11254.073} C_VEL
LIN {X 0,Y 395.831,Z 469.043,A -85,B 0,C 180,E1 -11255.807,E2 -11255.807} C_VEL
LIN {X 0,Y 396.054,Z 463.649,A -85,B 0,C 180,E1 -11257.647,E2 -11257.647} C_VEL
LIN {X 0,Y 396.394,Z 456.603,A -85,B 0,C 180,E1 -11259.438,E2 -11259.438} C_VEL
LIN {X 0,Y 396.833,Z 448.96,A -85,B 0,C 180,E1 -11260.974,E2 -11260.974} C_VEL
LIN {X 0,Y 397.462,Z 441.157,A -85,B 0,C 180,E1 -11262.249,E2 -11262.249} C_VEL
LIN {X 0,Y 398.249,Z 430.853,A -85,B 0,C 180,E1 -11263.613,E2 -11263.613} C_VEL
LIN {X 0,Y 398.986,Z 419.726,A -85,B 0,C 180,E1 -11264.796,E2 -11264.796} C_VEL
LIN {X 0,Y 399.689,Z 409.266,A -85,B 0,C 180,E1 -11265.683,E2 -11265.683} C_VEL
LIN {X 0,Y 400.524,Z 396.746,A -85,B 0,C 180,E1 -11266.5,E2 -11266.5} C_VEL
LIN {X 0,Y 401.195,Z 383.64,A -85,B 0,C 180,E1 -11267.126,E2 -11267.126} C_VEL
LIN {X 0,Y 401.704,Z 370.677,A -85,B 0,C 180,E1 -11267.531,E2 -11267.531} C_VEL
LIN {X 0,Y 402.824,Z 293.004,A -85,B 0,C 180,E1 -11269.036,E2 -11269.036} C_VEL
LIN {X 0,Y 398.659,Z 263.722,A -85,B 0,C 180,E1 -11269.835,E2 -11269.835} C_VEL
LIN {X 0,Y 400.015,Z 245.013,A -85,B 0,C 180,E1 -11273.557,E2 -11273.557} C_VEL
LIN {X 0,Y 400.496,Z 236.948,A -85,B 0,C 180,E1 -11275.182,E2 -11275.182} C_VEL
LIN {X 0,Y 398.045,Z 223.999,A -85,B 0,C 180,E1 -11278.015,E2 -11278.015} C_VEL
LIN {X 0,Y 397.156,Z 220.015,A -85,B 0,C 180,E1 -11278.971,E2 -11278.971} C_VEL
LIN {X 0,Y 397.067,Z 220.028,A -85,B 0,C 180,E1 -11282.068,E2 -11282.068} C_VEL
LIN {X 0,Y 397.105,Z 220.018,A -85,B 0,C 180,E1 -11285.5,E2 -11285.5} C_VEL
LIN {X 0,Y 397.111,Z 220.015,A -85,B 0,C 180,E1 -11288.857,E2 -11288.857} C_VEL
LIN {X 0,Y 397.048,Z 220.026,A -85,B 0,C 180,E1 -11292.264,E2 -11292.264} C_VEL
LIN {X 0,Y 397.064,Z 220.022,A -85,B 0,C 180,E1 -11295.066,E2 -11295.066} C_VEL
LIN {X 0,Y 397.04,Z 220.028,A -85,B 0,C 180,E1 -11298.018,E2 -11298.018} C_VEL
LIN {X 0,Y 397.097,Z 220.019,A -85,B 0,C 180,E1 -11301.137,E2 -11301.137} C_VEL
LIN {X 0,Y 397.089,Z 220.018,A -85,B 0,C 180,E1 -11304.494,E2 -11304.494} C_VEL
LIN {X 0,Y 397.045,Z 220.026,A -85,B 0,C 180,E1 -11307.925,E2 -11307.925} C_VEL
LIN {X 0,Y 397.081,Z 220.026,A -85,B 0,C 180,E1 -11311.453,E2 -11311.453} C_VEL
LIN {X 0,Y 397.116,Z 220.015,A -85,B 0,C 180,E1 -11314.485,E2 -11314.485} C_VEL
LIN {X 0,Y 397.055,Z 220.022,A -85,B 0,C 180,E1 -11318.179,E2 -11318.179} C_VEL
LIN {X 0,Y 397.119,Z 220.02,A -85,B 0,C 180,E1 -11321.424,E2 -11321.424} C_VEL
LIN {X 0,Y 397.135,Z 220.013,A -85,B 0,C 180,E1 -11324.606,E2 -11324.606} C_VEL
LIN {X 0,Y 397.185,Z 220.007,A -85,B 0,C 180,E1 -11327.74,E2 -11327.74} C_VEL
LIN {X 0,Y 397.285,Z 219.994,A -85,B 0,C 180,E1 -11331.864,E2 -11331.864} C_VEL
LIN {X 0,Y 397.321,Z 219.989,A -85,B 0,C 180,E1 -11333.907,E2 -11333.907} C_VEL
LIN {X 0,Y 397.4,Z 219.979,A -85,B 0,C 180,E1 -11337.973,E2 -11337.973} C_VEL
LIN {X 0,Y 397.53,Z 219.963,A -85,B 0,C 180,E1 -11340,E2 -11340} C_VEL
LIN {X 0,Y 397.328,Z 219.993,A -85,B 0,C 180,E1 -11343.041,E2 -11343.041} C_VEL
LIN {X 0,Y 397.317,Z 219.99,A -85,B 0,C 180,E1 -11346.763,E2 -11346.763} C_VEL
LIN {X 0,Y 397.209,Z 220.006,A -85,B 0,C 180,E1 -11349.162,E2 -11349.162} C_VEL
LIN {X 0,Y 397.186,Z 220.008,A -85,B 0,C 180,E1 -11352.259,E2 -11352.259} C_VEL
LIN {X 0,Y 397.139,Z 220.012,A -85,B 0,C 180,E1 -11355.393,E2 -11355.393} C_VEL
LIN {X 0,Y 397.131,Z 220.02,A -85,B 0,C 180,E1 -11358.575,E2 -11358.575} C_VEL
LIN {X 0,Y 397.148,Z 220.011,A -85,B 0,C 180,E1 -11361.815,E2 -11361.815} C_VEL
LIN {X 0,Y 397.115,Z 220.015,A -85,B 0,C 180,E1 -11365.514,E2 -11365.514} C_VEL
LIN {X 0,Y 397.089,Z 220.023,A -85,B 0,C 180,E1 -11368.546,E2 -11368.546} C_VEL
LIN {X 0,Y 397.044,Z 220.028,A -85,B 0,C 180,E1 -11372.074,E2 -11372.074} C_VEL
LIN {X 0,Y 397.087,Z 220.019,A -85,B 0,C 180,E1 -11375.506,E2 -11375.506} C_VEL
LIN {X 0,Y 397.108,Z 220.016,A -85,B 0,C 180,E1 -11378.865,E2 -11378.865} C_VEL
LIN {X 0,Y 397.13,Z 220.018,A -85,B 0,C 180,E1 -11382.259,E2 -11382.259} C_VEL
LIN {X 0,Y 397.08,Z 220.019,A -85,B 0,C 180,E1 -11385.069,E2 -11385.069} C_VEL
LIN {X 0,Y 397.064,Z 220.028,A -85,B 0,C 180,E1 -11388.021,E2 -11388.021} C_VEL
LIN {X 0,Y 397.116,Z 220.015,A -85,B 0,C 180,E1 -11391.141,E2 -11391.141} C_VEL
LIN {X 0,Y 397.102,Z 220.017,A -85,B 0,C 180,E1 -11394.5,E2 -11394.5} C_VEL
LIN {X 0,Y 397.066,Z 220.027,A -85,B 0,C 180,E1 -11397.931,E2 -11397.931} C_VEL
LIN {X 0,Y 397.114,Z 220.018,A -85,B 0,C 180,E1 -11401.459,E2 -11401.459} C_VEL
LIN {X 0,Y 397.142,Z 220.012,A -85,B 0,C 180,E1 -11404.49,E2 -11404.49} C_VEL
LIN {X 0,Y 397.1,Z 220.018,A -85,B 0,C 180,E1 -11407.088,E2 -11407.088} C_VEL
LIN {X 0,Y 397.141,Z 220.012,A -85,B 0,C 180,E1 -11410.355,E2 -11410.355} C_VEL
LIN {X 0,Y 397.161,Z 220.016,A -85,B 0,C 180,E1 -11413.555,E2 -11413.555} C_VEL
LIN {X 0,Y 397.224,Z 220.002,A -85,B 0,C 180,E1 -11416.704,E2 -11416.704} C_VEL
LIN {X 0,Y 397.215,Z 220.005,A -85,B 0,C 180,E1 -11419.81,E2 -11419.81} C_VEL
LIN {X 0,Y 397.347,Z 219.988,A -85,B 0,C 180,E1 -11422.889,E2 -11422.889} C_VEL
LIN {X 0,Y 397.251,Z 220.001,A -85,B 0,C 180,E1 -11424.926,E2 -11424.926} C_VEL
LIN {X 0,Y 397.449,Z 219.974,A -85,B 0,C 180,E1 -11427.974,E2 -11427.974} C_VEL
LIN {X 0,Y 397.578,Z 219.957,A -85,B 0,C 180,E1 -11430,E2 -11430} C_VEL
LIN {X 0,Y 397.38,Z 219.988,A -85,B 0,C 180,E1 -11433.041,E2 -11433.041} C_VEL
LIN {X 0,Y 397.36,Z 219.984,A -85,B 0,C 180,E1 -11436.091,E2 -11436.091} C_VEL
LIN {X 0,Y 397.249,Z 220.003,A -85,B 0,C 180,E1 -11439.161,E2 -11439.161} C_VEL
LIN {X 0,Y 397.216,Z 220.003,A -85,B 0,C 180,E1 -11442.257,E2 -11442.257} C_VEL
LIN {X 0,Y 397.174,Z 220.009,A -85,B 0,C 180,E1 -11445.391,E2 -11445.391} C_VEL
LIN {X 0,Y 397.156,Z 220.013,A -85,B 0,C 180,E1 -11448.572,E2 -11448.572} C_VEL
LIN {X 0,Y 397.081,Z 220.019,A -85,B 0,C 180,E1 -11451.954,E2 -11451.954} C_VEL
LIN {X 0,Y 397.143,Z 220.015,A -85,B 0,C 180,E1 -11455.51,E2 -11455.51} C_VEL
LIN {X 0,Y 397.124,Z 220.018,A -85,B 0,C 180,E1 -11456.366,E2 -11456.366} C_VEL
LIN {X 0,Y 396.485,Z 220.3,A -85,B 0,C 180,E1 -11456.939,E2 -11456.939} C_VEL
LIN {X 0,Y 395.024,Z 221.057,A -85,B 0,C 180,E1 -11457.48,E2 -11457.48} C_VEL
LIN {X 0,Y 391.827,Z 223.715,A -85,B 0,C 180,E1 -11458.511,E2 -11458.511} C_VEL
LIN {X 0,Y 391.139,Z 225.862,A -85,B 0,C 180,E1 -11459.115,E2 -11459.115} C_VEL
LIN {X 0,Y 391.186,Z 226.194,A -85,B 0,C 180,E1 -11459.201,E2 -11459.201} C_VEL
LIN {X 0,Y 391.813,Z 229.267,A -85,B 0,C 180,E1 -11459.959,E2 -11459.959} C_VEL
LIN {X 0,Y 393.881,Z 237.433,A -85,B 0,C 180,E1 -11460.228,E2 -11460.228} C_VEL
LIN {X 0,Y 396.509,Z 250.751,A -85,B 0,C 180,E1 -11460.627,E2 -11460.627} C_VEL
LIN {X 0,Y 394.976,Z 337.272,A -85,B 0,C 180,E1 -11462.347,E2 -11462.347} C_VEL
LIN {X 0,Y 394.505,Z 350.049,A -85,B 0,C 180,E1 -11462.796,E2 -11462.796} C_VEL
LIN {X 0,Y 394.02,Z 363.459,A -85,B 0,C 180,E1 -11463.499,E2 -11463.499} C_VEL
LIN {X 0,Y 393.359,Z 375.327,A -85,B 0,C 180,E1 -11464.344,E2 -11464.344} C_VEL
LIN {X 0,Y 392.577,Z 387.102,A -85,B 0,C 180,E1 -11465.417,E2 -11465.417} C_VEL
LIN {X 0,Y 391.834,Z 397.425,A -85,B 0,C 180,E1 -11466.606,E2 -11466.606} C_VEL
LIN {X 0,Y 390.985,Z 407.34,A -85,B 0,C 180,E1 -11468.023,E2 -11468.023} C_VEL
LIN {X 0,Y 390.377,Z 415.762,A -85,B 0,C 180,E1 -11469.518,E2 -11469.518} C_VEL
LIN {X 0,Y 389.826,Z 422.489,A -85,B 0,C 180,E1 -11471.001,E2 -11471.001} C_VEL
LIN {X 0,Y 389.393,Z 428.776,A -85,B 0,C 180,E1 -11472.755,E2 -11472.755} C_VEL
LIN {X 0,Y 389.128,Z 433.087,A -85,B 0,C 180,E1 -11474.313,E2 -11474.313} C_VEL
LIN {X 0,Y 388.86,Z 436.176,A -85,B 0,C 180,E1 -11475.788,E2 -11475.788} C_VEL
LIN {X 0,Y 388.662,Z 439.018,A -85,B 0,C 180,E1 -11477.843,E2 -11477.843} C_VEL
LIN {X 0,Y 388.6,Z 440.07,A -85,B 0,C 180,E1 -11479.421,E2 -11479.421} C_VEL
LIN {X 0,Y 388.595,Z 440.172,A -85,B 0,C 180,E1 -11481.041,E2 -11481.041} C_VEL
LIN {X 0,Y 388.701,Z 439.254,A -85,B 0,C 180,E1 -11482.699,E2 -11482.699} C_VEL
LIN {X 0,Y 388.941,Z 436.766,A -85,B 0,C 180,E1 -11484.675,E2 -11484.675} C_VEL
LIN {X 0,Y 389.183,Z 433.885,A -85,B 0,C 180,E1 -11486.16,E2 -11486.16} C_VEL
LIN {X 0,Y 389.696,Z 429.107,A -85,B 0,C 180,E1 -11487.944,E2 -11487.944} C_VEL
LIN {X 0,Y 390.306,Z 422.542,A -85,B 0,C 180,E1 -11489.793,E2 -11489.793} C_VEL
LIN {X 0,Y 391.046,Z 415.344,A -85,B 0,C 180,E1 -11491.361,E2 -11491.361} C_VEL
LIN {X 0,Y 391.849,Z 407.277,A -85,B 0,C 180,E1 -11492.784,E2 -11492.784} C_VEL
LIN {X 0,Y 392.686,Z 397.883,A -85,B 0,C 180,E1 -11494.136,E2 -11494.136} C_VEL
LIN {X 0,Y 393.518,Z 388.262,A -85,B 0,C 180,E1 -11495.257,E2 -11495.257} C_VEL
LIN {X 0,Y 394.418,Z 377.918,A -85,B 0,C 180,E1 -11496.225,E2 -11496.225} C_VEL
LIN {X 0,Y 395.251,Z 365.536,A -85,B 0,C 180,E1 -11497.14,E2 -11497.14} C_VEL
LIN {X 0,Y 395.928,Z 352.821,A -85,B 0,C 180,E1 -11497.839,E2 -11497.839} C_VEL
LIN {X 0,Y 396.377,Z 339.261,A -85,B 0,C 180,E1 -11498.345,E2 -11498.345} C_VEL
LIN {X 0,Y 397.105,Z 304.031,A -85,B 0,C 180,E1 -11499.084,E2 -11499.084} C_VEL
LIN {X 0,Y 398.173,Z 250.852,A -85,B 0,C 180,E1 -11500.166,E2 -11500.166} C_VEL
LIN {X 0,Y 395.016,Z 237.251,A -85,B 0,C 180,E1 -11500.671,E2 -11500.671} C_VEL
LIN {X 0,Y 392.147,Z 229.866,A -85,B 0,C 180,E1 -11501.058,E2 -11501.058} C_VEL
LIN {X 0,Y 390.128,Z 220.89,A -85,B 0,C 180,E1 -11503.248,E2 -11503.248} C_VEL
LIN {X 0,Y 390.154,Z 220.891,A -85,B 0,C 180,E1 -11506.561,E2 -11506.561} C_VEL
LIN {X 0,Y 390.131,Z 220.894,A -85,B 0,C 180,E1 -11509.622,E2 -11509.622} C_VEL
LIN {X 0,Y 390.266,Z 220.874,A -85,B 0,C 180,E1 -11512.759,E2 -11512.759} C_VEL
LIN {X 0,Y 390.187,Z 220.882,A -85,B 0,C 180,E1 -11514.833,E2 -11514.833} C_VEL
LIN {X 0,Y 390.37,Z 220.858,A -85,B 0,C 180,E1 -11517.937,E2 -11517.937} C_VEL
LIN {X 0,Y 390.501,Z 220.842,A -85,B 0,C 180,E1 -11520,E2 -11520} C_VEL
LIN {X 0,Y 390.262,Z 220.872,A -85,B 0,C 180,E1 -11523.097,E2 -11523.097} C_VEL
LIN {X 0,Y 390.276,Z 220.866,A -85,B 0,C 180,E1 -11526.203,E2 -11526.203} C_VEL
LIN {X 0,Y 390.163,Z 220.885,A -85,B 0,C 180,E1 -11529.33,E2 -11529.33} C_VEL
LIN {X 0,Y 390.135,Z 220.886,A -85,B 0,C 180,E1 -11532.485,E2 -11532.485} C_VEL
LIN {X 0,Y 390.1,Z 220.89,A -85,B 0,C 180,E1 -11535.679,E2 -11535.679} C_VEL
LIN {X 0,Y 390.06,Z 220.898,A -85,B 0,C 180,E1 -11538.925,E2 -11538.925} C_VEL
LIN {X 0,Y 389.999,Z 220.906,A -85,B 0,C 180,E1 -11542.237,E2 -11542.237} C_VEL
LIN {X 0,Y 390.084,Z 220.892,A -85,B 0,C 180,E1 -11545.745,E2 -11545.745} C_VEL
LIN {X 0,Y 390.019,Z 220.897,A -85,B 0,C 180,E1 -11549.113,E2 -11549.113} C_VEL
LIN {X 0,Y 390.012,Z 220.901,A -85,B 0,C 180,E1 -11552.725,E2 -11552.725} C_VEL
LIN {X 0,Y 390.027,Z 220.897,A -85,B 0,C 180,E1 -11555.828,E2 -11555.828} C_VEL
LIN {X 0,Y 390.035,Z 220.899,A -85,B 0,C 180,E1 -11559.22,E2 -11559.22} C_VEL
LIN {X 0,Y 390.017,Z 220.902,A -85,B 0,C 180,E1 -11562.377,E2 -11562.377} C_VEL
LIN {X 0,Y 390.023,Z 220.898,A -85,B 0,C 180,E1 -11565.357,E2 -11565.357} C_VEL
LIN {X 0,Y 390.012,Z 220.904,A -85,B 0,C 180,E1 -11568.19,E2 -11568.19} C_VEL
LIN {X 0,Y 390.072,Z 220.895,A -85,B 0,C 180,E1 -11570.911,E2 -11570.911} C_VEL
LIN {X 0,Y 390.072,Z 220.894,A -85,B 0,C 180,E1 -11574.796,E2 -11574.796} C_VEL
LIN {X 0,Y 390.013,Z 220.906,A -85,B 0,C 180,E1 -11578.499,E2 -11578.499} C_VEL
LIN {X 0,Y 390.096,Z 221.079,A -85,B 0,C 180,E1 -11580.527,E2 -11580.527} C_VEL
LIN {X 0,Y 392.727,Z 232.451,A -85,B 0,C 180,E1 -11583.141,E2 -11583.141} C_VEL
LIN {X 0,Y 393.87,Z 239.325,A -85,B 0,C 180,E1 -11584.647,E2 -11584.647} C_VEL
LIN {X 0,Y 392.863,Z 253.088,A -85,B 0,C 180,E1 -11587.383,E2 -11587.383} C_VEL
LIN {X 0,Y 392.267,Z 261.426,A -85,B 0,C 180,E1 -11589.023,E2 -11589.023} C_VEL
LIN {X 0,Y 396.085,Z 283.426,A -85,B 0,C 180,E1 -11589.756,E2 -11589.756} C_VEL
LIN {X 0,Y 397.506,Z 294.714,A -85,B 0,C 180,E1 -11590.086,E2 -11590.086} C_VEL
LIN {X 0,Y 396.116,Z 371.175,A -85,B 0,C 180,E1 -11591.646,E2 -11591.646} C_VEL
LIN {X 0,Y 395.371,Z 384.712,A -85,B 0,C 180,E1 -11592.112,E2 -11592.112} C_VEL
LIN {X 0,Y 394.545,Z 397.63,A -85,B 0,C 180,E1 -11592.776,E2 -11592.776} C_VEL
LIN {X 0,Y 393.517,Z 410.244,A -85,B 0,C 180,E1 -11593.665,E2 -11593.665} C_VEL
LIN {X 0,Y 392.54,Z 421.546,A -85,B 0,C 180,E1 -11594.689,E2 -11594.689} C_VEL
LIN {X 0,Y 391.7,Z 431.694,A -85,B 0,C 180,E1 -11595.84,E2 -11595.84} C_VEL
LIN {X 0,Y 390.959,Z 440.208,A -85,B 0,C 180,E1 -11597.016,E2 -11597.016} C_VEL
LIN {X 0,Y 390.027,Z 449.409,A -85,B 0,C 180,E1 -11598.569,E2 -11598.569} C_VEL
LIN {X 0,Y 389.447,Z 456.847,A -85,B 0,C 180,E1 -11600.13,E2 -11600.13} C_VEL
LIN {X 0,Y 389.063,Z 462.814,A -85,B 0,C 180,E1 -11601.692,E2 -11601.692} C_VEL
LIN {X 0,Y 388.825,Z 467.522,A -85,B 0,C 180,E1 -11603.254,E2 -11603.254} C_VEL
LIN {X 0,Y 388.724,Z 471.115,A -85,B 0,C 180,E1 -11604.814,E2 -11604.814} C_VEL
LIN {X 0,Y 388.704,Z 472.917,A -85,B 0,C 180,E1 -11605.853,E2 -11605.853} C_VEL
LIN {X 0,Y 388.755,Z 475.282,A -85,B 0,C 180,E1 -11607.928,E2 -11607.928} C_VEL
LIN {X 0,Y 388.762,Z 475.842,A -85,B 0,C 180,E1 -11608.964,E2 -11608.964} C_VEL
LIN {X 0,Y 388.751,Z 475.957,A -85,B 0,C 180,E1 -11610,E2 -11610} C_VEL
LIN {X 0,Y 388.762,Z 475.675,A -85,B 0,C 180,E1 -11611.036,E2 -11611.036} C_VEL
LIN {X 0,Y 388.787,Z 474.995,A -85,B 0,C 180,E1 -11612.072,E2 -11612.072} C_VEL
LIN {X 0,Y 388.679,Z 473.874,A -85,B 0,C 180,E1 -11613.109,E2 -11613.109} C_VEL
LIN {X 0,Y 388.726,Z 471.385,A -85,B 0,C 180,E1 -11614.666,E2 -11614.666} C_VEL
LIN {X 0,Y 388.795,Z 467.848,A -85,B 0,C 180,E1 -11616.226,E2 -11616.226} C_VEL
LIN {X 0,Y 388.982,Z 463.177,A -85,B 0,C 180,E1 -11617.787,E2 -11617.787} C_VEL
LIN {X 0,Y 389.335,Z 456.084,A -85,B 0,C 180,E1 -11619.611,E2 -11619.611} C_VEL
LIN {X 0,Y 389.828,Z 448.392,A -85,B 0,C 180,E1 -11621.174,E2 -11621.174} C_VEL
LIN {X 0,Y 390.462,Z 440.52,A -85,B 0,C 180,E1 -11622.472,E2 -11622.472} C_VEL
LIN {X 0,Y 391.223,Z 431.087,A -85,B 0,C 180,E1 -11623.744,E2 -11623.744} C_VEL
LIN {X 0,Y 391.972,Z 420.203,A -85,B 0,C 180,E1 -11624.934,E2 -11624.934} C_VEL
LIN {X 0,Y 392.819,Z 408.265,A -85,B 0,C 180,E1 -11625.965,E2 -11625.965} C_VEL
LIN {X 0,Y 393.645,Z 395.528,A -85,B 0,C 180,E1 -11626.796,E2 -11626.796} C_VEL
LIN {X 0,Y 394.364,Z 382.887,A -85,B 0,C 180,E1 -11627.399,E2 -11627.399} C_VEL
LIN {X 0,Y 394.887,Z 369.555,A -85,B 0,C 180,E1 -11627.81,E2 -11627.81} C_VEL
LIN {X 0,Y 395.958,Z 293.713,A -85,B 0,C 180,E1 -11629.311,E2 -11629.311} C_VEL
LIN {X 0,Y 391.72,Z 263.436,A -85,B 0,C 180,E1 -11630.159,E2 -11630.159} C_VEL
LIN {X 0,Y 393.073,Z 245.832,A -85,B 0,C 180,E1 -11633.719,E2 -11633.719} C_VEL
LIN {X 0,Y 393.504,Z 237.765,A -85,B 0,C 180,E1 -11635.378,E2 -11635.378} C_VEL
LIN {X 0,Y 391.006,Z 224.844,A -85,B 0,C 180,E1 -11638.268,E2 -11638.268} C_VEL
LIN {X 0,Y 390.094,Z 220.895,A -85,B 0,C 180,E1 -11639.214,E2 -11639.214} C_VEL
LIN {X 0,Y 390.031,Z 220.899,A -85,B 0,C 180,E1 -11642.718,E2 -11642.718} C_VEL
LIN {X 0,Y 390.042,Z 220.901,A -85,B 0,C 180,E1 -11645.822,E2 -11645.822} C_VEL
LIN {X 0,Y 390.051,Z 220.895,A -85,B 0,C 180,E1 -11649.214,E2 -11649.214} C_VEL
LIN {X 0,Y 390.022,Z 220.9,A -85,B 0,C 180,E1 -11652.37,E2 -11652.37} C_VEL
LIN {X 0,Y 390.022,Z 220.901,A -85,B 0,C 180,E1 -11655.351,E2 -11655.351} C_VEL
LIN {X 0,Y 390.005,Z 220.903,A -85,B 0,C 180,E1 -11658.183,E2 -11658.183} C_VEL
LIN {X 0,Y 390.056,Z 220.895,A -85,B 0,C 180,E1 -11660.903,E2 -11660.903} C_VEL
LIN {X 0,Y 390.055,Z 220.894,A -85,B 0,C 180,E1 -11664.79,E2 -11664.79} C_VEL
LIN {X 0,Y 389.989,Z 220.902,A -85,B 0,C 180,E1 -11668.492,E2 -11668.492} C_VEL
LIN {X 0,Y 390.084,Z 220.892,A -85,B 0,C 180,E1 -11672.067,E2 -11672.067} C_VEL
LIN {X 0,Y 390.04,Z 220.902,A -85,B 0,C 180,E1 -11675.516,E2 -11675.516} C_VEL
LIN {X 0,Y 390.033,Z 220.901,A -85,B 0,C 180,E1 -11679.534,E2 -11679.534} C_VEL
LIN {X 0,Y 390.096,Z 220.896,A -85,B 0,C 180,E1 -11683.246,E2 -11683.246} C_VEL
LIN {X 0,Y 390.154,Z 220.883,A -85,B 0,C 180,E1 -11686.56,E2 -11686.56} C_VEL
LIN {X 0,Y 390.129,Z 220.887,A -85,B 0,C 180,E1 -11689.621,E2 -11689.621} C_VEL
LIN {X 0,Y 390.253,Z 220.873,A -85,B 0,C 180,E1 -11692.758,E2 -11692.758} C_VEL
LIN {X 0,Y 390.175,Z 220.884,A -85,B 0,C 180,E1 -11694.832,E2 -11694.832} C_VEL
LIN {X 0,Y 390.369,Z 220.855,A -85,B 0,C 180,E1 -11697.936,E2 -11697.936} C_VEL
LIN {X 0,Y 390.5,Z 220.839,A -85,B 0,C 180,E1 -11700,E2 -11700} C_VEL
LIN {X 0,Y 390.263,Z 220.873,A -85,B 0,C 180,E1 -11703.097,E2 -11703.097} C_VEL
LIN {X 0,Y 390.269,Z 220.867,A -85,B 0,C 180,E1 -11706.76,E2 -11706.76} C_VEL
LIN {X 0,Y 390.162,Z 220.882,A -85,B 0,C 180,E1 -11709.329,E2 -11709.329} C_VEL
LIN {X 0,Y 390.135,Z 220.889,A -85,B 0,C 180,E1 -11712.484,E2 -11712.484} C_VEL
LIN {X 0,Y 390.099,Z 220.889,A -85,B 0,C 180,E1 -11715.678,E2 -11715.678} C_VEL
LIN {X 0,Y 390.08,Z 220.894,A -85,B 0,C 180,E1 -11718.923,E2 -11718.923} C_VEL
LIN {X 0,Y 390.086,Z 220.894,A -85,B 0,C 180,E1 -11722.231,E2 -11722.231} C_VEL
LIN {X 0,Y 390.081,Z 220.892,A -85,B 0,C 180,E1 -11725.745,E2 -11725.745} C_VEL
LIN {X 0,Y 390.027,Z 220.898,A -85,B 0,C 180,E1 -11729.112,E2 -11729.112} C_VEL
LIN {X 0,Y 390.009,Z 220.902,A -85,B 0,C 180,E1 -11732.724,E2 -11732.724} C_VEL
LIN {X 0,Y 390.025,Z 220.9,A -85,B 0,C 180,E1 -11735.828,E2 -11735.828} C_VEL
LIN {X 0,Y 390.045,Z 220.895,A -85,B 0,C 180,E1 -11739.222,E2 -11739.222} C_VEL
LIN {X 0,Y 390.092,Z 220.893,A -85,B 0,C 180,E1 -11742.389,E2 -11742.389} C_VEL
LIN {X 0,Y 390.033,Z 220.898,A -85,B 0,C 180,E1 -11745.359,E2 -11745.359} C_VEL
LIN {X 0,Y 390.055,Z 220.895,A -85,B 0,C 180,E1 -11749.178,E2 -11749.178} C_VEL
LIN {X 0,Y 390.028,Z 220.899,A -85,B 0,C 180,E1 -11752.452,E2 -11752.452} C_VEL
LIN {X 0,Y 390.052,Z 220.899,A -85,B 0,C 180,E1 -11756.048,E2 -11756.048} C_VEL
LIN {X 0,Y 390.038,Z 220.902,A -85,B 0,C 180,E1 -11759.871,E2 -11759.871} C_VEL
LIN {X 0,Y 390.102,Z 220.89,A -85,B 0,C 180,E1 -11763.234,E2 -11763.234} C_VEL
LIN {X 0,Y 390.098,Z 220.889,A -85,B 0,C 180,E1 -11766.753,E2 -11766.753} C_VEL
LIN {X 0,Y 390.1,Z 220.891,A -85,B 0,C 180,E1 -11769.985,E2 -11769.985} C_VEL
LIN {X 0,Y 390.133,Z 220.888,A -85,B 0,C 180,E1 -11773.25,E2 -11773.25} C_VEL
LIN {X 0,Y 390.19,Z 220.877,A -85,B 0,C 180,E1 -11776.563,E2 -11776.563} C_VEL
LIN {X 0,Y 390.202,Z 220.876,A -85,B 0,C 180,E1 -11780.672,E2 -11780.672} C_VEL
LIN {X 0,Y 390.322,Z 220.863,A -85,B 0,C 180,E1 -11783.799,E2 -11783.799} C_VEL
LIN {X 0,Y 390.418,Z 220.85,A -85,B 0,C 180,E1 -11787.937,E2 -11787.937} C_VEL
LIN {X 0,Y 390.547,Z 220.833,A -85,B 0,C 180,E1 -11790,E2 -11790} C_VEL
LIN {X 0,Y 390.313,Z 220.868,A -85,B 0,C 180,E1 -11793.096,E2 -11793.096} C_VEL
LIN {X 0,Y 390.313,Z 220.862,A -85,B 0,C 180,E1 -11796.202,E2 -11796.202} C_VEL
LIN {X 0,Y 390.202,Z 220.879,A -85,B 0,C 180,E1 -11799.328,E2 -11799.328} C_VEL
LIN {X 0,Y 390.191,Z 220.879,A -85,B 0,C 180,E1 -11803.437,E2 -11803.437} C_VEL
LIN {X 0,Y 390.143,Z 220.886,A -85,B 0,C 180,E1 -11807.306,E2 -11807.306} C_VEL
LIN {X 0,Y 390.08,Z 220.894,A -85,B 0,C 180,E1 -11810.468,E2 -11810.468} C_VEL
LIN {X 0,Y 390.065,Z 220.894,A -85,B 0,C 180,E1 -11813.35,E2 -11813.35} C_VEL
LIN {X 0,Y 390.101,Z 220.895,A -85,B 0,C 180,E1 -11816.766,E2 -11816.766} C_VEL
LIN {X 0,Y 390.157,Z 220.897,A -85,B 0,C 180,E1 -11817.851,E2 -11817.851} C_VEL
LIN {X 0,Y 391.186,Z 226.194,A -85,B 0,C 180,E1 -11819.201,E2 -11819.201} C_VEL
LIN {X 0,Y 391.459,Z 228.616,A -85,B 0,C 180,E1 -11819.592,E2 -11819.592} C_VEL
LIN {X 0,Y 391.538,Z 232.968,A -85,B 0,C 180,E1 -11819.924,E2 -11819.924} C_VEL
LIN {X 0,Y 391.275,Z 239.296,A -85,B 0,C 180,E1 -11820.133,E2 -11820.133} C_VEL
LIN {X 0,Y 389.648,Z 256.693,A -85,B 0,C 180,E1 -11820.436,E2 -11820.436} C_VEL
LIN {X 0,Y 388.147,Z 337.414,A -85,B 0,C 180,E1 -11822.072,E2 -11822.072} C_VEL
LIN {X 0,Y 387.656,Z 351.005,A -85,B 0,C 180,E1 -11822.564,E2 -11822.564} C_VEL
LIN {X 0,Y 387.121,Z 364.043,A -85,B 0,C 180,E1 -11823.267,E2 -11823.267} C_VEL
LIN {X 0,Y 386.379,Z 376.706,A -85,B 0,C 180,E1 -11824.196,E2 -11824.196} C_VEL
LIN {X 0,Y 385.59,Z 388.164,A -85,B 0,C 180,E1 -11825.279,E2 -11825.279} C_VEL
LIN {X 0,Y 384.793,Z 398.581,A -85,B 0,C 180,E1 -11826.522,E2 -11826.522} C_VEL
LIN {X 0,Y 384.014,Z 407.387,A -85,B 0,C 180,E1 -11827.809,E2 -11827.809} C_VEL
LIN {X 0,Y 383.385,Z 415.925,A -85,B 0,C 180,E1 -11829.342,E2 -11829.342} C_VEL
LIN {X 0,Y 382.803,Z 422.672,A -85,B 0,C 180,E1 -11830.847,E2 -11830.847} C_VEL
LIN {X 0,Y 382.34,Z 429.111,A -85,B 0,C 180,E1 -11832.671,E2 -11832.671} C_VEL
LIN {X 0,Y 382.052,Z 433.629,A -85,B 0,C 180,E1 -11834.343,E2 -11834.343} C_VEL
LIN {X 0,Y 381.76,Z 436.724,A -85,B 0,C 180,E1 -11835.881,E2 -11835.881} C_VEL
LIN {X 0,Y 381.601,Z 438.908,A -85,B 0,C 180,E1 -11837.443,E2 -11837.443} C_VEL
LIN {X 0,Y 381.512,Z 440.199,A -85,B 0,C 180,E1 -11839.043,E2 -11839.043} C_VEL
LIN {X 0,Y 381.508,Z 440.481,A -85,B 0,C 180,E1 -11841.22,E2 -11841.22} C_VEL
LIN {X 0,Y 381.615,Z 439.745,A -85,B 0,C 180,E1 -11842.574,E2 -11842.574} C_VEL
LIN {X 0,Y 381.785,Z 438.152,A -85,B 0,C 180,E1 -11844.084,E2 -11844.084} C_VEL
LIN {X 0,Y 382.046,Z 435.165,A -85,B 0,C 180,E1 -11845.865,E2 -11845.865} C_VEL
LIN {X 0,Y 382.601,Z 430.412,A -85,B 0,C 180,E1 -11847.812,E2 -11847.812} C_VEL
LIN {X 0,Y 383.153,Z 424.69,A -85,B 0,C 180,E1 -11849.542,E2 -11849.542} C_VEL
LIN {X 0,Y 383.913,Z 417.519,A -85,B 0,C 180,E1 -11851.24,E2 -11851.24} C_VEL
LIN {X 0,Y 384.85,Z 408.991,A -85,B 0,C 180,E1 -11852.836,E2 -11852.836} C_VEL
LIN {X 0,Y 385.727,Z 399.839,A -85,B 0,C 180,E1 -11854.215,E2 -11854.215} C_VEL
LIN {X 0,Y 386.678,Z 389.548,A -85,B 0,C 180,E1 -11855.469,E2 -11855.469} C_VEL
LIN {X 0,Y 387.631,Z 379.032,A -85,B 0,C 180,E1 -11856.493,E2 -11856.493} C_VEL
LIN {X 0,Y 388.452,Z 367.774,A -85,B 0,C 180,E1 -11857.359,E2 -11857.359} C_VEL
LIN {X 0,Y 389.15,Z 355.867,A -85,B 0,C 180,E1 -11858.062,E2 -11858.062} C_VEL
LIN {X 0,Y 389.666,Z 342.799,A -85,B 0,C 180,E1 -11858.613,E2 -11858.613} C_VEL
LIN {X 0,Y 390.076,Z 326.474,A -85,B 0,C 180,E1 -11859.016,E2 -11859.016} C_VEL
LIN {X 0,Y 391.748,Z 252.22,A -85,B 0,C 180,E1 -11860.553,E2 -11860.553} C_VEL
LIN {X 0,Y 388.904,Z 240.025,A -85,B 0,C 180,E1 -11861.018,E2 -11861.018} C_VEL
LIN {X 0,Y 385.053,Z 230.318,A -85,B 0,C 180,E1 -11861.525,E2 -11861.525} C_VEL
LIN {X 0,Y 383.084,Z 221.767,A -85,B 0,C 180,E1 -11863.685,E2 -11863.685} C_VEL
LIN {X 0,Y 383.1,Z 221.773,A -85,B 0,C 180,E1 -11867.283,E2 -11867.283} C_VEL
LIN {X 0,Y 383.11,Z 221.766,A -85,B 0,C 180,E1 -11870.497,E2 -11870.497} C_VEL
LIN {X 0,Y 383.25,Z 221.747,A -85,B 0,C 180,E1 -11873.683,E2 -11873.683} C_VEL
LIN {X 0,Y 383.338,Z 221.734,A -85,B 0,C 180,E1 -11877.899,E2 -11877.899} C_VEL
LIN {X 0,Y 383.471,Z 221.718,A -85,B 0,C 180,E1 -11880,E2 -11880} C_VEL
LIN {X 0,Y 383.198,Z 221.751,A -85,B 0,C 180,E1 -11883.154,E2 -11883.154} C_VEL
LIN {X 0,Y 383.233,Z 221.744,A -85,B 0,C 180,E1 -11886.318,E2 -11886.318} C_VEL
LIN {X 0,Y 383.181,Z 221.752,A -85,B 0,C 180,E1 -11888.438,E2 -11888.438} C_VEL
LIN {X 0,Y 383.063,Z 221.765,A -85,B 0,C 180,E1 -11891.644,E2 -11891.644} C_VEL
LIN {X 0,Y 383.071,Z 221.766,A -85,B 0,C 180,E1 -11894.884,E2 -11894.884} C_VEL
LIN {X 0,Y 383.022,Z 221.771,A -85,B 0,C 180,E1 -11898.176,E2 -11898.176} C_VEL
LIN {X 0,Y 382.953,Z 221.781,A -85,B 0,C 180,E1 -11901.534,E2 -11901.534} C_VEL
LIN {X 0,Y 383.015,Z 221.775,A -85,B 0,C 180,E1 -11904.963,E2 -11904.963} C_VEL
LIN {X 0,Y 382.995,Z 221.778,A -85,B 0,C 180,E1 -11908.272,E2 -11908.272} C_VEL
LIN {X 0,Y 382.977,Z 221.778,A -85,B 0,C 180,E1 -11912.153,E2 -11912.153} C_VEL
LIN {X 0,Y 382.99,Z 221.776,A -85,B 0,C 180,E1 -11914.671,E2 -11914.671} C_VEL
LIN {X 0,Y 382.97,Z 221.779,A -85,B 0,C 180,E1 -11917.906,E2 -11917.906} C_VEL
LIN {X 0,Y 382.955,Z 221.78,A -85,B 0,C 180,E1 -11921.352,E2 -11921.352} C_VEL
LIN {X 0,Y 382.974,Z 221.782,A -85,B 0,C 180,E1 -11924.306,E2 -11924.306} C_VEL
LIN {X 0,Y 382.993,Z 221.775,A -85,B 0,C 180,E1 -11927.244,E2 -11927.244} C_VEL
LIN {X 0,Y 382.998,Z 221.779,A -85,B 0,C 180,E1 -11930.417,E2 -11930.417} C_VEL
LIN {X 0,Y 383.011,Z 221.778,A -85,B 0,C 180,E1 -11934.048,E2 -11934.048} C_VEL
LIN {X 0,Y 382.976,Z 221.782,A -85,B 0,C 180,E1 -11937.581,E2 -11937.581} C_VEL
LIN {X 0,Y 383.033,Z 221.781,A -85,B 0,C 180,E1 -11940.071,E2 -11940.071} C_VEL
LIN {X 0,Y 385.503,Z 232.466,A -85,B 0,C 180,E1 -11942.595,E2 -11942.595} C_VEL
LIN {X 0,Y 386.996,Z 240.696,A -85,B 0,C 180,E1 -11944.452,E2 -11944.452} C_VEL
LIN {X 0,Y 386.076,Z 253.049,A -85,B 0,C 180,E1 -11946.962,E2 -11946.962} C_VEL
LIN {X 0,Y 385.435,Z 261.048,A -85,B 0,C 180,E1 -11948.563,E2 -11948.563} C_VEL
LIN {X 0,Y 389.429,Z 283.357,A -85,B 0,C 180,E1 -11949.334,E2 -11949.334} C_VEL
LIN {X 0,Y 390.946,Z 295.61,A -85,B 0,C 180,E1 -11949.705,E2 -11949.705} C_VEL
LIN {X 0,Y 389.467,Z 371.164,A -85,B 0,C 180,E1 -11951.287,E2 -11951.287} C_VEL
LIN {X 0,Y 388.638,Z 385.317,A -85,B 0,C 180,E1 -11951.792,E2 -11951.792} C_VEL
LIN {X 0,Y 387.795,Z 397.919,A -85,B 0,C 180,E1 -11952.467,E2 -11952.467} C_VEL
LIN {X 0,Y 386.73,Z 410.398,A -85,B 0,C 180,E1 -11953.37,E2 -11953.37} C_VEL
LIN {X 0,Y 385.681,Z 421.613,A -85,B 0,C 180,E1 -11954.41,E2 -11954.41} C_VEL
LIN {X 0,Y 384.739,Z 432.348,A -85,B 0,C 180,E1 -11955.672,E2 -11955.672} C_VEL
LIN {X 0,Y 383.862,Z 441.778,A -85,B 0,C 180,E1 -11957.041,E2 -11957.041} C_VEL
LIN {X 0,Y 382.901,Z 450.634,A -85,B 0,C 180,E1 -11958.621,E2 -11958.621} C_VEL
LIN {X 0,Y 382.344,Z 457.72,A -85,B 0,C 180,E1 -11960.212,E2 -11960.212} C_VEL
LIN {X 0,Y 381.896,Z 464.26,A -85,B 0,C 180,E1 -11962.067,E2 -11962.067} C_VEL
LIN {X 0,Y 381.654,Z 469.206,A -85,B 0,C 180,E1 -11963.93,E2 -11963.93} C_VEL
LIN {X 0,Y 381.627,Z 472.634,A -85,B 0,C 180,E1 -11965.776,E2 -11965.776} C_VEL
LIN {X 0,Y 381.654,Z 474.98,A -85,B 0,C 180,E1 -11967.89,E2 -11967.89} C_VEL
LIN {X 0,Y 381.693,Z 475.517,A -85,B 0,C 180,E1 -11968.945,E2 -11968.945} C_VEL
LIN {X 0,Y 381.68,Z 475.62,A -85,B 0,C 180,E1 -11970,E2 -11970} C_VEL
LIN {X 0,Y 381.694,Z 475.326,A -85,B 0,C 180,E1 -11971.055,E2 -11971.055} C_VEL
LIN {X 0,Y 381.685,Z 474.631,A -85,B 0,C 180,E1 -11972.11,E2 -11972.11} C_VEL
LIN {X 0,Y 381.586,Z 473.483,A -85,B 0,C 180,E1 -11973.167,E2 -11973.167} C_VEL
LIN {X 0,Y 381.643,Z 470.965,A -85,B 0,C 180,E1 -11974.753,E2 -11974.753} C_VEL
LIN {X 0,Y 381.71,Z 467.395,A -85,B 0,C 180,E1 -11976.342,E2 -11976.342} C_VEL
LIN {X 0,Y 381.903,Z 462.682,A -85,B 0,C 180,E1 -11977.932,E2 -11977.932} C_VEL
LIN {X 0,Y 382.213,Z 456.682,A -85,B 0,C 180,E1 -11979.524,E2 -11979.524} C_VEL
LIN {X 0,Y 382.698,Z 449.183,A -85,B 0,C 180,E1 -11981.116,E2 -11981.116} C_VEL
LIN {X 0,Y 383.365,Z 441.544,A -85,B 0,C 180,E1 -11982.438,E2 -11982.438} C_VEL
LIN {X 0,Y 384.123,Z 432.281,A -85,B 0,C 180,E1 -11983.758,E2 -11983.758} C_VEL
LIN {X 0,Y 384.858,Z 421.971,A -85,B 0,C 180,E1 -11984.946,E2 -11984.946} C_VEL
LIN {X 0,Y 385.689,Z 410.556,A -85,B 0,C 180,E1 -11985.996,E2 -11985.996} C_VEL
LIN {X 0,Y 386.602,Z 398.769,A -85,B 0,C 180,E1 -11986.84,E2 -11986.84} C_VEL
LIN {X 0,Y 387.276,Z 386.626,A -85,B 0,C 180,E1 -11987.489,E2 -11987.489} C_VEL
LIN {X 0,Y 387.875,Z 373.455,A -85,B 0,C 180,E1 -11987.972,E2 -11987.972} C_VEL
LIN {X 0,Y 388.484,Z 340.67,A -85,B 0,C 180,E1 -11988.66,E2 -11988.66} C_VEL
LIN {X 0,Y 389.091,Z 293.853,A -85,B 0,C 180,E1 -11989.608,E2 -11989.608} C_VEL
LIN {X 0,Y 384.803,Z 263.184,A -85,B 0,C 180,E1 -11990.477,E2 -11990.477} C_VEL
LIN {X 0,Y 386.33,Z 244.035,A -85,B 0,C 180,E1 -11994.43,E2 -11994.43} C_VEL
LIN {X 0,Y 386.487,Z 238.581,A -85,B 0,C 180,E1 -11995.584,E2 -11995.584} C_VEL
LIN {X 0,Y 383.728,Z 224.793,A -85,B 0,C 180,E1 -11998.732,E2 -11998.732} C_VEL
LIN {X 0,Y 383.058,Z 221.771,A -85,B 0,C 180,E1 -11999.464,E2 -11999.464} C_VEL
LIN {X 0,Y 382.992,Z 221.775,A -85,B 0,C 180,E1 -12003.398,E2 -12003.398} C_VEL
LIN {X 0,Y 383.018,Z 221.775,A -85,B 0,C 180,E1 -12006.161,E2 -12006.161} C_VEL
LIN {X 0,Y 382.991,Z 221.78,A -85,B 0,C 180,E1 -12009.955,E2 -12009.955} C_VEL
LIN {X 0,Y 382.987,Z 221.775,A -85,B 0,C 180,E1 -12012.775,E2 -12012.775} C_VEL
LIN {X 0,Y 382.975,Z 221.783,A -85,B 0,C 180,E1 -12015.785,E2 -12015.785} C_VEL
LIN {X 0,Y 382.962,Z 221.778,A -85,B 0,C 180,E1 -12018.793,E2 -12018.793} C_VEL
LIN {X 0,Y 382.97,Z 221.779,A -85,B 0,C 180,E1 -12022.094,E2 -12022.094} C_VEL
LIN {X 0,Y 382.989,Z 221.778,A -85,B 0,C 180,E1 -12025.329,E2 -12025.329} C_VEL
LIN {X 0,Y 382.949,Z 221.782,A -85,B 0,C 180,E1 -12029.078,E2 -12029.078} C_VEL
LIN {X 0,Y 383.022,Z 221.771,A -85,B 0,C 180,E1 -12032.695,E2 -12032.695} C_VEL
LIN {X 0,Y 383.014,Z 221.774,A -85,B 0,C 180,E1 -12035.037,E2 -12035.037} C_VEL
LIN {X 0,Y 382.952,Z 221.779,A -85,B 0,C 180,E1 -12038.466,E2 -12038.466} C_VEL
LIN {X 0,Y 383.013,Z 221.773,A -85,B 0,C 180,E1 -12041.824,E2 -12041.824} C_VEL
LIN {X 0,Y 383.067,Z 221.77,A -85,B 0,C 180,E1 -12045.116,E2 -12045.116} C_VEL
LIN {X 0,Y 383.062,Z 221.766,A -85,B 0,C 180,E1 -12048.356,E2 -12048.356} C_VEL
LIN {X 0,Y 383.219,Z 221.746,A -85,B 0,C 180,E1 -12051.977,E2 -12051.977} C_VEL
LIN {X 0,Y 383.148,Z 221.758,A -85,B 0,C 180,E1 -12054.737,E2 -12054.737} C_VEL
LIN {X 0,Y 383.337,Z 221.731,A -85,B 0,C 180,E1 -12057.898,E2 -12057.898} C_VEL
LIN {X 0,Y 383.47,Z 221.715,A -85,B 0,C 180,E1 -12060,E2 -12060} C_VEL
LIN {X 0,Y 383.2,Z 221.752,A -85,B 0,C 180,E1 -12063.154,E2 -12063.154} C_VEL
LIN {X 0,Y 383.225,Z 221.745,A -85,B 0,C 180,E1 -12066.753,E2 -12066.753} C_VEL
LIN {X 0,Y 383.109,Z 221.76,A -85,B 0,C 180,E1 -12069.503,E2 -12069.503} C_VEL
LIN {X 0,Y 383.099,Z 221.767,A -85,B 0,C 180,E1 -12072.717,E2 -12072.717} C_VEL
LIN {X 0,Y 383.041,Z 221.769,A -85,B 0,C 180,E1 -12075.975,E2 -12075.975} C_VEL
LIN {X 0,Y 383.038,Z 221.769,A -85,B 0,C 180,E1 -12079.284,E2 -12079.284} C_VEL
LIN {X 0,Y 383.028,Z 221.774,A -85,B 0,C 180,E1 -12082.663,E2 -12082.663} C_VEL
LIN {X 0,Y 383.043,Z 221.771,A -85,B 0,C 180,E1 -12086.126,E2 -12086.126} C_VEL
LIN {X 0,Y 383.007,Z 221.778,A -85,B 0,C 180,E1 -12088.495,E2 -12088.495} C_VEL
LIN {X 0,Y 382.975,Z 221.781,A -85,B 0,C 180,E1 -12092.152,E2 -12092.152} C_VEL
LIN {X 0,Y 382.986,Z 221.777,A -85,B 0,C 180,E1 -12094.671,E2 -12094.671} C_VEL
LIN {X 0,Y 382.973,Z 221.78,A -85,B 0,C 180,E1 -12097.907,E2 -12097.907} C_VEL
LIN {X 0,Y 383.019,Z 221.771,A -85,B 0,C 180,E1 -12101.342,E2 -12101.342} C_VEL
LIN {X 0,Y 383.005,Z 221.777,A -85,B 0,C 180,E1 -12104.311,E2 -12104.311} C_VEL
LIN {X 0,Y 382.988,Z 221.775,A -85,B 0,C 180,E1 -12107.243,E2 -12107.243} C_VEL
LIN {X 0,Y 383.001,Z 221.775,A -85,B 0,C 180,E1 -12110.416,E2 -12110.416} C_VEL
LIN {X 0,Y 383.009,Z 221.777,A -85,B 0,C 180,E1 -12114.047,E2 -12114.047} C_VEL
LIN {X 0,Y 382.973,Z 221.78,A -85,B 0,C 180,E1 -12117.581,E2 -12117.581} C_VEL
LIN {X 0,Y 382.984,Z 221.777,A -85,B 0,C 180,E1 -12120.303,E2 -12120.303} C_VEL
LIN {X 0,Y 383.045,Z 221.767,A -85,B 0,C 180,E1 -12122.701,E2 -12122.701} C_VEL
LIN {X 0,Y 383.024,Z 221.772,A -85,B 0,C 180,E1 -12126.195,E2 -12126.195} C_VEL
LIN {X 0,Y 383.053,Z 221.773,A -85,B 0,C 180,E1 -12129.601,E2 -12129.601} C_VEL
LIN {X 0,Y 383.099,Z 221.762,A -85,B 0,C 180,E1 -12132.933,E2 -12132.933} C_VEL
LIN {X 0,Y 383.121,Z 221.758,A -85,B 0,C 180,E1 -12136.465,E2 -12136.465} C_VEL
LIN {X 0,Y 383.149,Z 221.755,A -85,B 0,C 180,E1 -12140.499,E2 -12140.499} C_VEL
LIN {X 0,Y 383.278,Z 221.741,A -85,B 0,C 180,E1 -12143.684,E2 -12143.684} C_VEL
LIN {X 0,Y 383.386,Z 221.726,A -85,B 0,C 180,E1 -12147.899,E2 -12147.899} C_VEL
LIN {X 0,Y 383.516,Z 221.709,A -85,B 0,C 180,E1 -12150,E2 -12150} C_VEL
LIN {X 0,Y 383.25,Z 221.749,A -85,B 0,C 180,E1 -12153.153,E2 -12153.153} C_VEL
LIN {X 0,Y 383.27,Z 221.74,A -85,B 0,C 180,E1 -12156.316,E2 -12156.316} C_VEL
LIN {X 0,Y 383.22,Z 221.747,A -85,B 0,C 180,E1 -12158.436,E2 -12158.436} C_VEL
LIN {X 0,Y 383.094,Z 221.762,A -85,B 0,C 180,E1 -12161.641,E2 -12161.641} C_VEL
LIN {X 0,Y 383.105,Z 221.766,A -85,B 0,C 180,E1 -12164.88,E2 -12164.88} C_VEL
LIN {X 0,Y 383.057,Z 221.767,A -85,B 0,C 180,E1 -12168.172,E2 -12168.172} C_VEL
LIN {X 0,Y 382.984,Z 221.775,A -85,B 0,C 180,E1 -12171.529,E2 -12171.529} C_VEL
LIN {X 0,Y 383.042,Z 221.774,A -85,B 0,C 180,E1 -12174.958,E2 -12174.958} C_VEL
LIN {X 0,Y 383.142,Z 221.923,A -85,B 0,C 180,E1 -12177.662,E2 -12177.662} C_VEL
LIN {X 0,Y 384.604,Z 229.396,A -85,B 0,C 180,E1 -12179.597,E2 -12179.597} C_VEL
LIN {X 0,Y 386.907,Z 237.101,A -85,B 0,C 180,E1 -12179.89,E2 -12179.89} C_VEL
LIN {X 0,Y 389.685,Z 251.403,A -85,B 0,C 180,E1 -12180.327,E2 -12180.327} C_VEL
LIN {X 0,Y 389.648,Z 256.693,A -85,B 0,C 180,E1 -12180.436,E2 -12180.436} C_VEL
LIN {X 0,Y 388.988,Z 262.52,A -85,B 0,C 180,E1 -12180.526,E2 -12180.526} C_VEL
LIN {X 0,Y 383.139,Z 281.456,A -85,B 0,C 180,E1 -12180.657,E2 -12180.657} C_VEL
LIN {X 0,Y 382.276,Z 287.29,A -85,B 0,C 180,E1 -12180.742,E2 -12180.742} C_VEL
LIN {X 0,Y 381.314,Z 337.94,A -85,B 0,C 180,E1 -12181.8,E2 -12181.8} C_VEL
LIN {X 0,Y 380.788,Z 351.503,A -85,B 0,C 180,E1 -12182.302,E2 -12182.302} C_VEL
LIN {X 0,Y 380.28,Z 363.521,A -85,B 0,C 180,E1 -12182.955,E2 -12182.955} C_VEL
LIN {X 0,Y 379.602,Z 375.345,A -85,B 0,C 180,E1 -12183.816,E2 -12183.816} C_VEL
LIN {X 0,Y 378.728,Z 387.482,A -85,B 0,C 180,E1 -12184.951,E2 -12184.951} C_VEL
LIN {X 0,Y 377.912,Z 397.91,A -85,B 0,C 180,E1 -12186.188,E2 -12186.188} C_VEL
LIN {X 0,Y 377.02,Z 407.92,A -85,B 0,C 180,E1 -12187.666,E2 -12187.666} C_VEL
LIN {X 0,Y 376.374,Z 416.01,A -85,B 0,C 180,E1 -12189.145,E2 -12189.145} C_VEL
LIN {X 0,Y 375.711,Z 423.634,A -85,B 0,C 180,E1 -12190.892,E2 -12190.892} C_VEL
LIN {X 0,Y 375.256,Z 429.854,A -85,B 0,C 180,E1 -12192.718,E2 -12192.718} C_VEL
LIN {X 0,Y 374.916,Z 434.627,A -85,B 0,C 180,E1 -12194.576,E2 -12194.576} C_VEL
LIN {X 0,Y 374.64,Z 437.389,A -85,B 0,C 180,E1 -12196.045,E2 -12196.045} C_VEL
LIN {X 0,Y 374.5,Z 439.304,A -85,B 0,C 180,E1 -12197.501,E2 -12197.501} C_VEL
LIN {X 0,Y 374.446,Z 440.464,A -85,B 0,C 180,E1 -12198.935,E2 -12198.935} C_VEL
LIN {X 0,Y 374.409,Z 440.914,A -85,B 0,C 180,E1 -12200.342,E2 -12200.342} C_VEL
LIN {X 0,Y 374.47,Z 440.519,A -85,B 0,C 180,E1 -12202.014,E2 -12202.014} C_VEL
LIN {X 0,Y 374.661,Z 439.069,A -85,B 0,C 180,E1 -12203.757,E2 -12203.757} C_VEL
LIN {X 0,Y 374.964,Z 435.97,A -85,B 0,C 180,E1 -12205.786,E2 -12205.786} C_VEL
LIN {X 0,Y 375.409,Z 432.4,A -85,B 0,C 180,E1 -12207.389,E2 -12207.389} C_VEL
LIN {X 0,Y 376.023,Z 426.77,A -85,B 0,C 180,E1 -12209.279,E2 -12209.279} C_VEL
LIN {X 0,Y 376.752,Z 420.168,A -85,B 0,C 180,E1 -12210.987,E2 -12210.987} C_VEL
LIN {X 0,Y 377.62,Z 412.736,A -85,B 0,C 180,E1 -12212.512,E2 -12212.512} C_VEL
LIN {X 0,Y 378.574,Z 403.877,A -85,B 0,C 180,E1 -12213.987,E2 -12213.987} C_VEL
LIN {X 0,Y 379.505,Z 394.212,A -85,B 0,C 180,E1 -12215.296,E2 -12215.296} C_VEL
LIN {X 0,Y 380.438,Z 384.722,A -85,B 0,C 180,E1 -12216.339,E2 -12216.339} C_VEL
LIN {X 0,Y 381.474,Z 372.752,A -85,B 0,C 180,E1 -12217.382,E2 -12217.382} C_VEL
LIN {X 0,Y 382.294,Z 360.357,A -85,B 0,C 180,E1 -12218.216,E2 -12218.216} C_VEL
LIN {X 0,Y 382.915,Z 347.729,A -85,B 0,C 180,E1 -12218.828,E2 -12218.828} C_VEL
LIN {X 0,Y 383.38,Z 334.222,A -85,B 0,C 180,E1 -12219.25,E2 -12219.25} C_VEL
LIN {X 0,Y 385.137,Z 252.825,A -85,B 0,C 180,E1 -12220.98,E2 -12220.98} C_VEL
LIN {X 0,Y 382.752,Z 242.604,A -85,B 0,C 180,E1 -12221.382,E2 -12221.382} C_VEL
LIN {X 0,Y 377.938,Z 230.773,A -85,B 0,C 180,E1 -12222.028,E2 -12222.028} C_VEL
LIN {X 0,Y 376.022,Z 222.649,A -85,B 0,C 180,E1 -12224.137,E2 -12224.137} C_VEL
LIN {X 0,Y 376.073,Z 222.647,A -85,B 0,C 180,E1 -12227.041,E2 -12227.041} C_VEL
LIN {X 0,Y 376.079,Z 222.642,A -85,B 0,C 180,E1 -12230.318,E2 -12230.318} C_VEL
LIN {X 0,Y 376.207,Z 222.624,A -85,B 0,C 180,E1 -12233.565,E2 -12233.565} C_VEL
LIN {X 0,Y 376.305,Z 222.611,A -85,B 0,C 180,E1 -12237.86,E2 -12237.86} C_VEL
LIN {X 0,Y 376.442,Z 222.594,A -85,B 0,C 180,E1 -12240,E2 -12240} C_VEL
LIN {X 0,Y 376.136,Z 222.631,A -85,B 0,C 180,E1 -12243.214,E2 -12243.214} C_VEL
LIN {X 0,Y 376.192,Z 222.621,A -85,B 0,C 180,E1 -12246.436,E2 -12246.436} C_VEL
LIN {X 0,Y 376.079,Z 222.638,A -85,B 0,C 180,E1 -12249.683,E2 -12249.683} C_VEL
LIN {X 0,Y 376.051,Z 222.638,A -85,B 0,C 180,E1 -12253.659,E2 -12253.659} C_VEL
LIN {X 0,Y 376.005,Z 222.643,A -85,B 0,C 180,E1 -12257.608,E2 -12257.608} C_VEL
LIN {X 0,Y 375.944,Z 222.654,A -85,B 0,C 180,E1 -12260.835,E2 -12260.835} C_VEL
LIN {X 0,Y 375.953,Z 222.65,A -85,B 0,C 180,E1 -12264.285,E2 -12264.285} C_VEL
LIN {X 0,Y 375.987,Z 222.647,A -85,B 0,C 180,E1 -12266.655,E2 -12266.655} C_VEL
LIN {X 0,Y 375.932,Z 222.654,A -85,B 0,C 180,E1 -12270.316,E2 -12270.316} C_VEL
LIN {X 0,Y 375.932,Z 222.658,A -85,B 0,C 180,E1 -12274.115,E2 -12274.115} C_VEL
LIN {X 0,Y 375.926,Z 222.659,A -85,B 0,C 180,E1 -12276.745,E2 -12276.745} C_VEL
LIN {X 0,Y 375.951,Z 222.656,A -85,B 0,C 180,E1 -12279.971,E2 -12279.971} C_VEL
LIN {X 0,Y 375.908,Z 222.657,A -85,B 0,C 180,E1 -12283.77,E2 -12283.77} C_VEL
LIN {X 0,Y 375.916,Z 222.658,A -85,B 0,C 180,E1 -12286.814,E2 -12286.814} C_VEL
LIN {X 0,Y 375.946,Z 222.657,A -85,B 0,C 180,E1 -12290.54,E2 -12290.54} C_VEL
LIN {X 0,Y 375.95,Z 222.654,A -85,B 0,C 180,E1 -12293.499,E2 -12293.499} C_VEL
LIN {X 0,Y 375.949,Z 222.658,A -85,B 0,C 180,E1 -12295.892,E2 -12295.892} C_VEL
LIN {X 0,Y 375.971,Z 222.778,A -85,B 0,C 180,E1 -12299.657,E2 -12299.657} C_VEL
LIN {X 0,Y 378.331,Z 232.478,A -85,B 0,C 180,E1 -12302.031,E2 -12302.031} C_VEL
LIN {X 0,Y 379.942,Z 240.72,A -85,B 0,C 180,E1 -12303.943,E2 -12303.943} C_VEL
LIN {X 0,Y 379.982,Z 245.635,A -85,B 0,C 180,E1 -12304.998,E2 -12304.998} C_VEL
LIN {X 0,Y 378.666,Z 260.612,A -85,B 0,C 180,E1 -12308.071,E2 -12308.071} C_VEL
LIN {X 0,Y 382.867,Z 283.964,A -85,B 0,C 180,E1 -12308.917,E2 -12308.917} C_VEL
LIN {X 0,Y 384.415,Z 297.115,A -85,B 0,C 180,E1 -12309.32,E2 -12309.32} C_VEL
LIN {X 0,Y 382.9,Z 370.27,A -85,B 0,C 180,E1 -12310.884,E2 -12310.884} C_VEL
LIN {X 0,Y 382.088,Z 383.791,A -85,B 0,C 180,E1 -12311.364,E2 -12311.364} C_VEL
LIN {X 0,Y 381.273,Z 396.171,A -85,B 0,C 180,E1 -12312.018,E2 -12312.018} C_VEL
LIN {X 0,Y 380.253,Z 407.382,A -85,B 0,C 180,E1 -12312.801,E2 -12312.801} C_VEL
LIN {X 0,Y 379.106,Z 419.078,A -85,B 0,C 180,E1 -12313.856,E2 -12313.856} C_VEL
LIN {X 0,Y 378.066,Z 429.853,A -85,B 0,C 180,E1 -12315.08,E2 -12315.08} C_VEL
LIN {X 0,Y 377.202,Z 438.331,A -85,B 0,C 180,E1 -12316.259,E2 -12316.259} C_VEL
LIN {X 0,Y 376.42,Z 446.358,A -85,B 0,C 180,E1 -12317.603,E2 -12317.603} C_VEL
LIN {X 0,Y 375.553,Z 454.214,A -85,B 0,C 180,E1 -12319.215,E2 -12319.215} C_VEL
LIN {X 0,Y 375.073,Z 460.546,A -85,B 0,C 180,E1 -12320.836,E2 -12320.836} C_VEL
LIN {X 0,Y 374.747,Z 465.592,A -85,B 0,C 180,E1 -12322.457,E2 -12322.457} C_VEL
LIN {X 0,Y 374.575,Z 469.225,A -85,B 0,C 180,E1 -12323.947,E2 -12323.947} C_VEL
LIN {X 0,Y 374.551,Z 472.355,A -85,B 0,C 180,E1 -12325.696,E2 -12325.696} C_VEL
LIN {X 0,Y 374.552,Z 474.678,A -85,B 0,C 180,E1 -12327.849,E2 -12327.849} C_VEL
LIN {X 0,Y 374.624,Z 475.192,A -85,B 0,C 180,E1 -12328.925,E2 -12328.925} C_VEL
LIN {X 0,Y 374.611,Z 475.285,A -85,B 0,C 180,E1 -12330,E2 -12330} C_VEL
LIN {X 0,Y 374.626,Z 474.978,A -85,B 0,C 180,E1 -12331.075,E2 -12331.075} C_VEL
LIN {X 0,Y 374.584,Z 474.266,A -85,B 0,C 180,E1 -12332.15,E2 -12332.15} C_VEL
LIN {X 0,Y 374.498,Z 473.092,A -85,B 0,C 180,E1 -12333.227,E2 -12333.227} C_VEL
LIN {X 0,Y 374.561,Z 470.543,A -85,B 0,C 180,E1 -12334.843,E2 -12334.843} C_VEL
LIN {X 0,Y 374.631,Z 466.938,A -85,B 0,C 180,E1 -12336.462,E2 -12336.462} C_VEL
LIN {X 0,Y 374.845,Z 462.187,A -85,B 0,C 180,E1 -12338.083,E2 -12338.083} C_VEL
LIN {X 0,Y 375.246,Z 455.005,A -85,B 0,C 180,E1 -12339.975,E2 -12339.975} C_VEL
LIN {X 0,Y 375.843,Z 447.193,A -85,B 0,C 180,E1 -12341.595,E2 -12341.595} C_VEL
LIN {X 0,Y 376.464,Z 439.173,A -85,B 0,C 180,E1 -12342.944,E2 -12342.944} C_VEL
LIN {X 0,Y 377.396,Z 428.773,A -85,B 0,C 180,E1 -12344.362,E2 -12344.362} C_VEL
LIN {X 0,Y 378.121,Z 418.523,A -85,B 0,C 180,E1 -12345.495,E2 -12345.495} C_VEL
LIN {X 0,Y 378.962,Z 407.984,A -85,B 0,C 180,E1 -12346.426,E2 -12346.426} C_VEL
LIN {X 0,Y 379.861,Z 395.355,A -85,B 0,C 180,E1 -12347.286,E2 -12347.286} C_VEL
LIN {X 0,Y 380.668,Z 382.129,A -85,B 0,C 180,E1 -12347.942,E2 -12347.942} C_VEL
LIN {X 0,Y 381.203,Z 368.735,A -85,B 0,C 180,E1 -12348.367,E2 -12348.367} C_VEL
LIN {X 0,Y 382.334,Z 294.828,A -85,B 0,C 180,E1 -12349.893,E2 -12349.893} C_VEL
LIN {X 0,Y 377.904,Z 262.863,A -85,B 0,C 180,E1 -12350.822,E2 -12350.822} C_VEL
LIN {X 0,Y 379.519,Z 243.69,A -85,B 0,C 180,E1 -12354.852,E2 -12354.852} C_VEL
LIN {X 0,Y 379.431,Z 239.341,A -85,B 0,C 180,E1 -12355.8,E2 -12355.8} C_VEL
LIN {X 0,Y 376.864,Z 226.551,A -85,B 0,C 180,E1 -12358.778,E2 -12358.778} C_VEL
LIN {X 0,Y 375.974,Z 222.653,A -85,B 0,C 180,E1 -12359.767,E2 -12359.767} C_VEL
LIN {X 0,Y 375.938,Z 222.655,A -85,B 0,C 180,E1 -12362.825,E2 -12362.825} C_VEL
LIN {X 0,Y 375.944,Z 222.653,A -85,B 0,C 180,E1 -12365.412,E2 -12365.412} C_VEL
LIN {X 0,Y 375.957,Z 222.653,A -85,B 0,C 180,E1 -12368.267,E2 -12368.267} C_VEL
LIN {X 0,Y 375.915,Z 222.659,A -85,B 0,C 180,E1 -12371.597,E2 -12371.597} C_VEL
LIN {X 0,Y 375.905,Z 222.659,A -85,B 0,C 180,E1 -12375.265,E2 -12375.265} C_VEL
LIN {X 0,Y 375.91,Z 222.657,A -85,B 0,C 180,E1 -12378.396,E2 -12378.396} C_VEL
LIN {X 0,Y 375.943,Z 222.658,A -85,B 0,C 180,E1 -12381.727,E2 -12381.727} C_VEL
LIN {X 0,Y 375.951,Z 222.655,A -85,B 0,C 180,E1 -12385.33,E2 -12385.33} C_VEL
LIN {X 0,Y 375.907,Z 222.657,A -85,B 0,C 180,E1 -12388.433,E2 -12388.433} C_VEL
LIN {X 0,Y 375.948,Z 222.652,A -85,B 0,C 180,E1 -12392.137,E2 -12392.137} C_VEL
LIN {X 0,Y 375.969,Z 222.649,A -85,B 0,C 180,E1 -12394.536,E2 -12394.536} C_VEL
LIN {X 0,Y 375.918,Z 222.656,A -85,B 0,C 180,E1 -12398.043,E2 -12398.043} C_VEL
LIN {X 0,Y 375.961,Z 222.655,A -85,B 0,C 180,E1 -12401.47,E2 -12401.47} C_VEL
LIN {X 0,Y 376.016,Z 222.646,A -85,B 0,C 180,E1 -12404.83,E2 -12404.83} C_VEL
LIN {X 0,Y 376.014,Z 222.643,A -85,B 0,C 180,E1 -12408.135,E2 -12408.135} C_VEL
LIN {X 0,Y 376.175,Z 222.623,A -85,B 0,C 180,E1 -12411.921,E2 -12411.921} C_VEL
LIN {X 0,Y 376.12,Z 222.633,A -85,B 0,C 180,E1 -12414.639,E2 -12414.639} C_VEL
LIN {X 0,Y 376.304,Z 222.607,A -85,B 0,C 180,E1 -12417.859,E2 -12417.859} C_VEL
LIN {X 0,Y 376.44,Z 222.59,A -85,B 0,C 180,E1 -12420,E2 -12420} C_VEL
LIN {X 0,Y 376.138,Z 222.631,A -85,B 0,C 180,E1 -12423.213,E2 -12423.213} C_VEL
LIN {X 0,Y 376.187,Z 222.622,A -85,B 0,C 180,E1 -12426.743,E2 -12426.743} C_VEL
LIN {X 0,Y 376.078,Z 222.635,A -85,B 0,C 180,E1 -12429.682,E2 -12429.682} C_VEL
LIN {X 0,Y 376.049,Z 222.639,A -85,B 0,C 180,E1 -12433.658,E2 -12433.658} C_VEL
LIN {X 0,Y 376.005,Z 222.645,A -85,B 0,C 180,E1 -12437.609,E2 -12437.609} C_VEL
LIN {X 0,Y 376.004,Z 222.648,A -85,B 0,C 180,E1 -12440.859,E2 -12440.859} C_VEL
LIN {X 0,Y 375.966,Z 222.654,A -85,B 0,C 180,E1 -12444.283,E2 -12444.283} C_VEL
LIN {X 0,Y 375.984,Z 222.651,A -85,B 0,C 180,E1 -12446.654,E2 -12446.654} C_VEL
LIN {X 0,Y 375.938,Z 222.653,A -85,B 0,C 180,E1 -12449.081,E2 -12449.081} C_VEL
LIN {X 0,Y 375.917,Z 222.657,A -85,B 0,C 180,E1 -12452.831,E2 -12452.831} C_VEL
LIN {X 0,Y 375.926,Z 222.654,A -85,B 0,C 180,E1 -12455.418,E2 -12455.418} C_VEL
LIN {X 0,Y 375.948,Z 222.657,A -85,B 0,C 180,E1 -12458.274,E2 -12458.274} C_VEL
LIN {X 0,Y 375.963,Z 222.651,A -85,B 0,C 180,E1 -12461.613,E2 -12461.613} C_VEL
LIN {X 0,Y 375.942,Z 222.653,A -85,B 0,C 180,E1 -12465.266,E2 -12465.266} C_VEL
LIN {X 0,Y 375.954,Z 222.651,A -85,B 0,C 180,E1 -12469.14,E2 -12469.14} C_VEL
LIN {X 0,Y 375.948,Z 222.658,A -85,B 0,C 180,E1 -12471.915,E2 -12471.915} C_VEL
LIN {X 0,Y 375.964,Z 222.651,A -85,B 0,C 180,E1 -12475.336,E2 -12475.336} C_VEL
LIN {X 0,Y 375.945,Z 222.653,A -85,B 0,C 180,E1 -12478.441,E2 -12478.441} C_VEL
LIN {X 0,Y 375.991,Z 222.649,A -85,B 0,C 180,E1 -12482.144,E2 -12482.144} C_VEL
LIN {X 0,Y 375.996,Z 222.646,A -85,B 0,C 180,E1 -12484.541,E2 -12484.541} C_VEL
LIN {X 0,Y 375.957,Z 222.653,A -85,B 0,C 180,E1 -12488.048,E2 -12488.048} C_VEL
LIN {X 0,Y 376.018,Z 222.649,A -85,B 0,C 180,E1 -12491.476,E2 -12491.476} C_VEL
LIN {X 0,Y 376.054,Z 222.639,A -85,B 0,C 180,E1 -12494.834,E2 -12494.834} C_VEL
LIN {X 0,Y 376.046,Z 222.64,A -85,B 0,C 180,E1 -12498.138,E2 -12498.138} C_VEL
LIN {X 0,Y 376.216,Z 222.62,A -85,B 0,C 180,E1 -12501.92,E2 -12501.92} C_VEL
LIN {X 0,Y 376.167,Z 222.625,A -85,B 0,C 180,E1 -12504.641,E2 -12504.641} C_VEL
LIN {X 0,Y 376.352,Z 222.602,A -85,B 0,C 180,E1 -12507.86,E2 -12507.86} C_VEL
LIN {X 0,Y 376.486,Z 222.585,A -85,B 0,C 180,E1 -12510,E2 -12510} C_VEL
LIN {X 0,Y 376.188,Z 222.628,A -85,B 0,C 180,E1 -12513.213,E2 -12513.213} C_VEL
LIN {X 0,Y 376.228,Z 222.618,A -85,B 0,C 180,E1 -12516.435,E2 -12516.435} C_VEL
LIN {X 0,Y 376.116,Z 222.631,A -85,B 0,C 180,E1 -12519.681,E2 -12519.681} C_VEL
LIN {X 0,Y 376.085,Z 222.635,A -85,B 0,C 180,E1 -12523.656,E2 -12523.656} C_VEL
LIN {X 0,Y 376.038,Z 222.641,A -85,B 0,C 180,E1 -12527.605,E2 -12527.605} C_VEL
LIN {X 0,Y 375.971,Z 222.655,A -85,B 0,C 180,E1 -12530.83,E2 -12530.83} C_VEL
LIN {X 0,Y 375.981,Z 222.65,A -85,B 0,C 180,E1 -12534.28,E2 -12534.28} C_VEL
LIN {X 0,Y 376.073,Z 222.664,A -85,B 0,C 180,E1 -12537.396,E2 -12537.396} C_VEL
LIN {X 0,Y 377.454,Z 229.719,A -85,B 0,C 180,E1 -12539.26,E2 -12539.26} C_VEL
LIN {X 0,Y 380.402,Z 239.478,A -85,B 0,C 180,E1 -12539.625,E2 -12539.625} C_VEL
LIN {X 0,Y 382.93,Z 253.165,A -85,B 0,C 180,E1 -12540.042,E2 -12540.042} C_VEL
LIN {X 0,Y 382.276,Z 287.29,A -85,B 0,C 180,E1 -12540.742,E2 -12540.742} C_VEL
LIN {X 0,Y 381.451,Z 293.113,A -85,B 0,C 180,E1 -12540.829,E2 -12540.829} C_VEL
LIN {X 0,Y 375.698,Z 312.051,A -85,B 0,C 180,E1 -12540.977,E2 -12540.977} C_VEL
LIN {X 0,Y 374.876,Z 317.876,A -85,B 0,C 180,E1 -12541.066,E2 -12541.066} C_VEL
LIN {X 0,Y 374.384,Z 339.57,A -85,B 0,C 180,E1 -12541.56,E2 -12541.56} C_VEL
LIN {X 0,Y 373.921,Z 352.431,A -85,B 0,C 180,E1 -12542.062,E2 -12542.062} C_VEL
LIN {X 0,Y 373.409,Z 363.789,A -85,B 0,C 180,E1 -12542.695,E2 -12542.695} C_VEL
LIN {X 0,Y 372.698,Z 375.487,A -85,B 0,C 180,E1 -12543.559,E2 -12543.559} C_VEL
LIN {X 0,Y 371.797,Z 387.58,A -85,B 0,C 180,E1 -12544.707,E2 -12544.707} C_VEL
LIN {X 0,Y 370.971,Z 398.017,A -85,B 0,C 180,E1 -12545.96,E2 -12545.96} C_VEL
LIN {X 0,Y 370.088,Z 407.768,A -85,B 0,C 180,E1 -12547.417,E2 -12547.417} C_VEL
LIN {X 0,Y 369.416,Z 415.747,A -85,B 0,C 180,E1 -12548.884,E2 -12548.884} C_VEL
LIN {X 0,Y 368.764,Z 422.435,A -85,B 0,C 180,E1 -12550.384,E2 -12550.384} C_VEL
LIN {X 0,Y 368.256,Z 429.079,A -85,B 0,C 180,E1 -12552.272,E2 -12552.272} C_VEL
LIN {X 0,Y 367.868,Z 434.304,A -85,B 0,C 180,E1 -12554.241,E2 -12554.241} C_VEL
LIN {X 0,Y 367.609,Z 437.247,A -85,B 0,C 180,E1 -12555.749,E2 -12555.749} C_VEL
LIN {X 0,Y 367.376,Z 440.092,A -85,B 0,C 180,E1 -12557.967,E2 -12557.967} C_VEL
LIN {X 0,Y 367.297,Z 441.161,A -85,B 0,C 180,E1 -12559.933,E2 -12559.933} C_VEL
LIN {X 0,Y 367.352,Z 441.037,A -85,B 0,C 180,E1 -12561.657,E2 -12561.657} C_VEL
LIN {X 0,Y 367.57,Z 439.637,A -85,B 0,C 180,E1 -12563.65,E2 -12563.65} C_VEL
LIN {X 0,Y 367.901,Z 436.573,A -85,B 0,C 180,E1 -12565.81,E2 -12565.81} C_VEL
LIN {X 0,Y 368.432,Z 432.389,A -85,B 0,C 180,E1 -12567.717,E2 -12567.717} C_VEL
LIN {X 0,Y 369.101,Z 426.478,A -85,B 0,C 180,E1 -12569.697,E2 -12569.697} C_VEL
LIN {X 0,Y 369.849,Z 420.207,A -85,B 0,C 180,E1 -12571.312,E2 -12571.312} C_VEL
LIN {X 0,Y 370.856,Z 412.274,A -85,B 0,C 180,E1 -12572.947,E2 -12572.947} C_VEL
LIN {X 0,Y 371.855,Z 403.296,A -85,B 0,C 180,E1 -12574.446,E2 -12574.446} C_VEL
LIN {X 0,Y 372.761,Z 394.516,A -85,B 0,C 180,E1 -12575.643,E2 -12575.643} C_VEL
LIN {X 0,Y 373.955,Z 383.214,A -85,B 0,C 180,E1 -12576.874,E2 -12576.874} C_VEL
LIN {X 0,Y 374.954,Z 371.945,A -85,B 0,C 180,E1 -12577.845,E2 -12577.845} C_VEL
LIN {X 0,Y 375.688,Z 360.671,A -85,B 0,C 180,E1 -12578.607,E2 -12578.607} C_VEL
LIN {X 0,Y 376.372,Z 347.767,A -85,B 0,C 180,E1 -12579.238,E2 -12579.238} C_VEL
LIN {X 0,Y 376.831,Z 334.547,A -85,B 0,C 180,E1 -12579.657,E2 -12579.657} C_VEL
LIN {X 0,Y 378.76,Z 254.238,A -85,B 0,C 180,E1 -12581.396,E2 -12581.396} C_VEL
LIN {X 0,Y 376.459,Z 244.661,A -85,B 0,C 180,E1 -12581.795,E2 -12581.795} C_VEL
LIN {X 0,Y 370.818,Z 231.194,A -85,B 0,C 180,E1 -12582.561,E2 -12582.561} C_VEL
LIN {X 0,Y 368.987,Z 223.526,A -85,B 0,C 180,E1 -12584.606,E2 -12584.606} C_VEL
LIN {X 0,Y 368.973,Z 223.531,A -85,B 0,C 180,E1 -12587.906,E2 -12587.906} C_VEL
LIN {X 0,Y 369.126,Z 223.507,A -85,B 0,C 180,E1 -12591.869,E2 -12591.869} C_VEL
LIN {X 0,Y 369.105,Z 223.508,A -85,B 0,C 180,E1 -12594.537,E2 -12594.537} C_VEL
LIN {X 0,Y 369.271,Z 223.487,A -85,B 0,C 180,E1 -12597.819,E2 -12597.819} C_VEL
LIN {X 0,Y 369.412,Z 223.469,A -85,B 0,C 180,E1 -12600,E2 -12600} C_VEL
LIN {X 0,Y 369.27,Z 223.487,A -85,B 0,C 180,E1 -12602.182,E2 -12602.182} C_VEL
LIN {X 0,Y 369.152,Z 223.499,A -85,B 0,C 180,E1 -12606.56,E2 -12606.56} C_VEL
LIN {X 0,Y 369.028,Z 223.516,A -85,B 0,C 180,E1 -12609.87,E2 -12609.87} C_VEL
LIN {X 0,Y 368.999,Z 223.516,A -85,B 0,C 180,E1 -12613.773,E2 -12613.773} C_VEL
LIN {X 0,Y 368.966,Z 223.52,A -85,B 0,C 180,E1 -12617.77,E2 -12617.77} C_VEL
LIN {X 0,Y 368.874,Z 223.536,A -85,B 0,C 180,E1 -12621.223,E2 -12621.223} C_VEL
LIN {X 0,Y 368.92,Z 223.533,A -85,B 0,C 180,E1 -12624.778,E2 -12624.778} C_VEL
LIN {X 0,Y 368.93,Z 223.527,A -85,B 0,C 180,E1 -12627.207,E2 -12627.207} C_VEL
LIN {X 0,Y 368.882,Z 223.535,A -85,B 0,C 180,E1 -12630.99,E2 -12630.99} C_VEL
LIN {X 0,Y 368.908,Z 223.528,A -85,B 0,C 180,E1 -12634.857,E2 -12634.857} C_VEL
LIN {X 0,Y 368.877,Z 223.536,A -85,B 0,C 180,E1 -12638.642,E2 -12638.642} C_VEL
LIN {X 0,Y 368.857,Z 223.54,A -85,B 0,C 180,E1 -12642.012,E2 -12642.012} C_VEL
LIN {X 0,Y 368.859,Z 223.535,A -85,B 0,C 180,E1 -12645.179,E2 -12645.179} C_VEL
LIN {X 0,Y 368.865,Z 223.537,A -85,B 0,C 180,E1 -12648.181,E2 -12648.181} C_VEL
LIN {X 0,Y 368.892,Z 223.534,A -85,B 0,C 180,E1 -12651.364,E2 -12651.364} C_VEL
LIN {X 0,Y 368.925,Z 223.529,A -85,B 0,C 180,E1 -12655.15,E2 -12655.15} C_VEL
LIN {X 0,Y 368.908,Z 223.585,A -85,B 0,C 180,E1 -12659.167,E2 -12659.167} C_VEL
LIN {X 0,Y 371.446,Z 233.939,A -85,B 0,C 180,E1 -12661.773,E2 -12661.773} C_VEL
LIN {X 0,Y 373.071,Z 242.119,A -85,B 0,C 180,E1 -12663.727,E2 -12663.727} C_VEL
LIN {X 0,Y 373.201,Z 246.429,A -85,B 0,C 180,E1 -12664.679,E2 -12664.679} C_VEL
LIN {X 0,Y 371.917,Z 260.223,A -85,B 0,C 180,E1 -12667.563,E2 -12667.563} C_VEL
LIN {X 0,Y 376.273,Z 284.138,A -85,B 0,C 180,E1 -12668.469,E2 -12668.469} C_VEL
LIN {X 0,Y 377.916,Z 297.455,A -85,B 0,C 180,E1 -12668.897,E2 -12668.897} C_VEL
LIN {X 0,Y 376.341,Z 369.595,A -85,B 0,C 180,E1 -12670.467,E2 -12670.467} C_VEL
LIN {X 0,Y 375.516,Z 383.203,A -85,B 0,C 180,E1 -12670.955,E2 -12670.955} C_VEL
LIN {X 0,Y 374.639,Z 395.635,A -85,B 0,C 180,E1 -12671.618,E2 -12671.618} C_VEL
LIN {X 0,Y 373.508,Z 407.678,A -85,B 0,C 180,E1 -12672.481,E2 -12672.481} C_VEL
LIN {X 0,Y 372.31,Z 419.225,A -85,B 0,C 180,E1 -12673.553,E2 -12673.553} C_VEL
LIN {X 0,Y 371.168,Z 430.223,A -85,B 0,C 180,E1 -12674.84,E2 -12674.84} C_VEL
LIN {X 0,Y 370.146,Z 439.971,A -85,B 0,C 180,E1 -12676.272,E2 -12676.272} C_VEL
LIN {X 0,Y 369.149,Z 449.04,A -85,B 0,C 180,E1 -12677.913,E2 -12677.913} C_VEL
LIN {X 0,Y 368.401,Z 456.347,A -85,B 0,C 180,E1 -12679.56,E2 -12679.56} C_VEL
LIN {X 0,Y 367.891,Z 462.188,A -85,B 0,C 180,E1 -12681.21,E2 -12681.21} C_VEL
LIN {X 0,Y 367.595,Z 466.806,A -85,B 0,C 180,E1 -12682.862,E2 -12682.862} C_VEL
LIN {X 0,Y 367.449,Z 470.325,A -85,B 0,C 180,E1 -12684.513,E2 -12684.513} C_VEL
LIN {X 0,Y 367.455,Z 472.087,A -85,B 0,C 180,E1 -12685.613,E2 -12685.613} C_VEL
LIN {X 0,Y 367.408,Z 473.435,A -85,B 0,C 180,E1 -12686.711,E2 -12686.711} C_VEL
LIN {X 0,Y 367.452,Z 474.377,A -85,B 0,C 180,E1 -12687.808,E2 -12687.808} C_VEL
LIN {X 0,Y 367.539,Z 474.868,A -85,B 0,C 180,E1 -12688.904,E2 -12688.904} C_VEL
LIN {X 0,Y 367.545,Z 474.947,A -85,B 0,C 180,E1 -12690,E2 -12690} C_VEL
LIN {X 0,Y 367.56,Z 474.627,A -85,B 0,C 180,E1 -12691.095,E2 -12691.095} C_VEL
LIN {X 0,Y 367.484,Z 473.894,A -85,B 0,C 180,E1 -12692.192,E2 -12692.192} C_VEL
LIN {X 0,Y 367.413,Z 472.696,A -85,B 0,C 180,E1 -12693.289,E2 -12693.289} C_VEL
LIN {X 0,Y 367.48,Z 470.115,A -85,B 0,C 180,E1 -12694.936,E2 -12694.936} C_VEL
LIN {X 0,Y 367.564,Z 466.474,A -85,B 0,C 180,E1 -12696.587,E2 -12696.587} C_VEL
LIN {X 0,Y 367.781,Z 461.681,A -85,B 0,C 180,E1 -12698.239,E2 -12698.239} C_VEL
LIN {X 0,Y 368.206,Z 454.451,A -85,B 0,C 180,E1 -12700.168,E2 -12700.168} C_VEL
LIN {X 0,Y 368.85,Z 446.556,A -85,B 0,C 180,E1 -12701.818,E2 -12701.818} C_VEL
LIN {X 0,Y 369.704,Z 436.659,A -85,B 0,C 180,E1 -12703.464,E2 -12703.464} C_VEL
LIN {X 0,Y 370.487,Z 427.815,A -85,B 0,C 180,E1 -12704.657,E2 -12704.657} C_VEL
LIN {X 0,Y 371.263,Z 417.607,A -85,B 0,C 180,E1 -12705.788,E2 -12705.788} C_VEL
LIN {X 0,Y 372.143,Z 406.875,A -85,B 0,C 180,E1 -12706.736,E2 -12706.736} C_VEL
LIN {X 0,Y 373.037,Z 394.023,A -85,B 0,C 180,E1 -12707.613,E2 -12707.613} C_VEL
LIN {X 0,Y 373.846,Z 381.142,A -85,B 0,C 180,E1 -12708.245,E2 -12708.245} C_VEL
LIN {X 0,Y 374.377,Z 367.322,A -85,B 0,C 180,E1 -12708.679,E2 -12708.679} C_VEL
LIN {X 0,Y 375.555,Z 295.725,A -85,B 0,C 180,E1 -12710.184,E2 -12710.184} C_VEL
LIN {X 0,Y 370.981,Z 262.652,A -85,B 0,C 180,E1 -12711.15,E2 -12711.15} C_VEL
LIN {X 0,Y 372.605,Z 244.105,A -85,B 0,C 180,E1 -12715.126,E2 -12715.126} C_VEL
LIN {X 0,Y 372.375,Z 240.115,A -85,B 0,C 180,E1 -12716.025,E2 -12716.025} C_VEL
LIN {X 0,Y 369.798,Z 227.403,A -85,B 0,C 180,E1 -12719.045,E2 -12719.045} C_VEL
LIN {X 0,Y 368.943,Z 223.53,A -85,B 0,C 180,E1 -12719.999,E2 -12719.999} C_VEL
LIN {X 0,Y 368.885,Z 223.533,A -85,B 0,C 180,E1 -12723.535,E2 -12723.535} C_VEL
LIN {X 0,Y 368.887,Z 223.531,A -85,B 0,C 180,E1 -12726.852,E2 -12726.852} C_VEL
LIN {X 0,Y 368.893,Z 223.532,A -85,B 0,C 180,E1 -12730.367,E2 -12730.367} C_VEL
LIN {X 0,Y 368.863,Z 223.538,A -85,B 0,C 180,E1 -12733.612,E2 -12733.612} C_VEL
LIN {X 0,Y 368.863,Z 223.534,A -85,B 0,C 180,E1 -12736.692,E2 -12736.692} C_VEL
LIN {X 0,Y 368.886,Z 223.537,A -85,B 0,C 180,E1 -12739.64,E2 -12739.64} C_VEL
LIN {X 0,Y 368.872,Z 223.535,A -85,B 0,C 180,E1 -12743.142,E2 -12743.142} C_VEL
LIN {X 0,Y 368.867,Z 223.534,A -85,B 0,C 180,E1 -12746.458,E2 -12746.458} C_VEL
LIN {X 0,Y 368.87,Z 223.534,A -85,B 0,C 180,E1 -12750.305,E2 -12750.305} C_VEL
LIN {X 0,Y 368.965,Z 223.523,A -85,B 0,C 180,E1 -12754.017,E2 -12754.017} C_VEL
LIN {X 0,Y 368.884,Z 223.535,A -85,B 0,C 180,E1 -12757.601,E2 -12757.601} C_VEL
LIN {X 0,Y 368.91,Z 223.533,A -85,B 0,C 180,E1 -12761.103,E2 -12761.103} C_VEL
LIN {X 0,Y 368.955,Z 223.523,A -85,B 0,C 180,E1 -12764.533,E2 -12764.533} C_VEL
LIN {X 0,Y 368.969,Z 223.521,A -85,B 0,C 180,E1 -12767.905,E2 -12767.905} C_VEL
LIN {X 0,Y 369.122,Z 223.502,A -85,B 0,C 180,E1 -12771.872,E2 -12771.872} C_VEL
LIN {X 0,Y 369.094,Z 223.507,A -85,B 0,C 180,E1 -12774.536,E2 -12774.536} C_VEL
LIN {X 0,Y 369.269,Z 223.484,A -85,B 0,C 180,E1 -12777.818,E2 -12777.818} C_VEL
LIN {X 0,Y 369.39,Z 223.469,A -85,B 0,C 180,E1 -12780,E2 -12780} C_VEL
LIN {X 0,Y 369.27,Z 223.484,A -85,B 0,C 180,E1 -12782.181,E2 -12782.181} C_VEL
LIN {X 0,Y 369.154,Z 223.5,A -85,B 0,C 180,E1 -12786.73,E2 -12786.73} C_VEL
LIN {X 0,Y 369.027,Z 223.514,A -85,B 0,C 180,E1 -12789.869,E2 -12789.869} C_VEL
LIN {X 0,Y 368.997,Z 223.518,A -85,B 0,C 180,E1 -12793.773,E2 -12793.773} C_VEL
LIN {X 0,Y 368.963,Z 223.522,A -85,B 0,C 180,E1 -12797.77,E2 -12797.77} C_VEL
LIN {X 0,Y 368.951,Z 223.524,A -85,B 0,C 180,E1 -12801.218,E2 -12801.218} C_VEL
LIN {X 0,Y 368.926,Z 223.529,A -85,B 0,C 180,E1 -12804.777,E2 -12804.777} C_VEL
LIN {X 0,Y 368.946,Z 223.53,A -85,B 0,C 180,E1 -12808.438,E2 -12808.438} C_VEL
LIN {X 0,Y 368.865,Z 223.54,A -85,B 0,C 180,E1 -12812.241,E2 -12812.241} C_VEL
LIN {X 0,Y 368.898,Z 223.53,A -85,B 0,C 180,E1 -12815.004,E2 -12815.004} C_VEL
LIN {X 0,Y 368.884,Z 223.534,A -85,B 0,C 180,E1 -12818.644,E2 -12818.644} C_VEL
LIN {X 0,Y 368.926,Z 223.532,A -85,B 0,C 180,E1 -12822.024,E2 -12822.024} C_VEL
LIN {X 0,Y 368.896,Z 223.53,A -85,B 0,C 180,E1 -12825.185,E2 -12825.185} C_VEL
LIN {X 0,Y 368.873,Z 223.538,A -85,B 0,C 180,E1 -12828.182,E2 -12828.182} C_VEL
LIN {X 0,Y 368.893,Z 223.532,A -85,B 0,C 180,E1 -12831.362,E2 -12831.362} C_VEL
LIN {X 0,Y 368.92,Z 223.528,A -85,B 0,C 180,E1 -12835.149,E2 -12835.149} C_VEL
LIN {X 0,Y 368.916,Z 223.528,A -85,B 0,C 180,E1 -12839.049,E2 -12839.049} C_VEL
LIN {X 0,Y 368.975,Z 223.525,A -85,B 0,C 180,E1 -12841.567,E2 -12841.567} C_VEL
LIN {X 0,Y 368.948,Z 223.526,A -85,B 0,C 180,E1 -12845.227,E2 -12845.227} C_VEL
LIN {X 0,Y 368.93,Z 223.527,A -85,B 0,C 180,E1 -12848.975,E2 -12848.975} C_VEL
LIN {X 0,Y 368.985,Z 223.52,A -85,B 0,C 180,E1 -12852.259,E2 -12852.259} C_VEL
LIN {X 0,Y 369.033,Z 223.513,A -85,B 0,C 180,E1 -12856.229,E2 -12856.229} C_VEL
LIN {X 0,Y 369.065,Z 223.51,A -85,B 0,C 180,E1 -12860.133,E2 -12860.133} C_VEL
LIN {X 0,Y 369.159,Z 223.497,A -85,B 0,C 180,E1 -12862.343,E2 -12862.343} C_VEL
LIN {X 0,Y 369.14,Z 223.5,A -85,B 0,C 180,E1 -12864.538,E2 -12864.538} C_VEL
LIN {X 0,Y 369.317,Z 223.479,A -85,B 0,C 180,E1 -12867.819,E2 -12867.819} C_VEL
LIN {X 0,Y 369.455,Z 223.461,A -85,B 0,C 180,E1 -12870,E2 -12870} C_VEL
LIN {X 0,Y 369.318,Z 223.478,A -85,B 0,C 180,E1 -12872.181,E2 -12872.181} C_VEL
LIN {X 0,Y 369.189,Z 223.495,A -85,B 0,C 180,E1 -12876.558,E2 -12876.558} C_VEL
LIN {X 0,Y 369.104,Z 223.508,A -85,B 0,C 180,E1 -12878.761,E2 -12878.761} C_VEL
LIN {X 0,Y 369.002,Z 223.517,A -85,B 0,C 180,E1 -12882.092,E2 -12882.092} C_VEL
LIN {X 0,Y 368.993,Z 223.519,A -85,B 0,C 180,E1 -12885.463,E2 -12885.463} C_VEL
LIN {X 0,Y 368.952,Z 223.529,A -85,B 0,C 180,E1 -12888.892,E2 -12888.892} C_VEL
LIN {X 0,Y 368.917,Z 223.53,A -85,B 0,C 180,E1 -12892.394,E2 -12892.394} C_VEL
LIN {X 0,Y 368.985,Z 223.523,A -85,B 0,C 180,E1 -12895.978,E2 -12895.978} C_VEL
LIN {X 0,Y 369.045,Z 223.695,A -85,B 0,C 180,E1 -12897.194,E2 -12897.194} C_VEL
LIN {X 0,Y 370.289,Z 230.182,A -85,B 0,C 180,E1 -12898.909,E2 -12898.909} C_VEL
LIN {X 0,Y 373.784,Z 241.139,A -85,B 0,C 180,E1 -12899.333,E2 -12899.333} C_VEL
LIN {X 0,Y 376.17,Z 254.114,A -85,B 0,C 180,E1 -12899.741,E2 -12899.741} C_VEL
LIN {X 0,Y 374.876,Z 317.876,A -85,B 0,C 180,E1 -12901.066,E2 -12901.066} C_VEL
LIN {X 0,Y 374.04,Z 323.71,A -85,B 0,C 180,E1 -12901.152,E2 -12901.152} C_VEL
LIN {X 0,Y 368.627,Z 340.675,A -85,B 0,C 180,E1 -12901.346,E2 -12901.346} C_VEL
LIN {X 0,Y 367.433,Z 346.363,A -85,B 0,C 180,E1 -12901.504,E2 -12901.504} C_VEL
LIN {X 0,Y 367.262,Z 348.263,A -85,B 0,C 180,E1 -12901.578,E2 -12901.578} C_VEL
LIN {X 0,Y 366.723,Z 360.474,A -85,B 0,C 180,E1 -12902.205,E2 -12902.205} C_VEL
LIN {X 0,Y 365.972,Z 373.24,A -85,B 0,C 180,E1 -12903.096,E2 -12903.096} C_VEL
LIN {X 0,Y 365.11,Z 384.697,A -85,B 0,C 180,E1 -12904.137,E2 -12904.137} C_VEL
LIN {X 0,Y 364.276,Z 395.332,A -85,B 0,C 180,E1 -12905.361,E2 -12905.361} C_VEL
LIN {X 0,Y 363.364,Z 405.67,A -85,B 0,C 180,E1 -12906.836,E2 -12906.836} C_VEL
LIN {X 0,Y 362.558,Z 414.107,A -85,B 0,C 180,E1 -12908.333,E2 -12908.333} C_VEL
LIN {X 0,Y 361.89,Z 421.092,A -85,B 0,C 180,E1 -12909.851,E2 -12909.851} C_VEL
LIN {X 0,Y 361.374,Z 426.866,A -85,B 0,C 180,E1 -12911.388,E2 -12911.388} C_VEL
LIN {X 0,Y 360.929,Z 432.825,A -85,B 0,C 180,E1 -12913.419,E2 -12913.419} C_VEL
LIN {X 0,Y 360.576,Z 437.102,A -85,B 0,C 180,E1 -12915.439,E2 -12915.439} C_VEL
LIN {X 0,Y 360.348,Z 439.355,A -85,B 0,C 180,E1 -12916.952,E2 -12916.952} C_VEL
LIN {X 0,Y 360.249,Z 440.778,A -85,B 0,C 180,E1 -12918.449,E2 -12918.449} C_VEL
LIN {X 0,Y 360.22,Z 441.482,A -85,B 0,C 180,E1 -12919.922,E2 -12919.922} C_VEL
LIN {X 0,Y 360.26,Z 441.505,A -85,B 0,C 180,E1 -12921.373,E2 -12921.373} C_VEL
LIN {X 0,Y 360.384,Z 440.623,A -85,B 0,C 180,E1 -12923.08,E2 -12923.08} C_VEL
LIN {X 0,Y 360.668,Z 438.611,A -85,B 0,C 180,E1 -12924.918,E2 -12924.918} C_VEL
LIN {X 0,Y 361.132,Z 434.927,A -85,B 0,C 180,E1 -12926.982,E2 -12926.982} C_VEL
LIN {X 0,Y 361.722,Z 430.545,A -85,B 0,C 180,E1 -12928.737,E2 -12928.737} C_VEL
LIN {X 0,Y 362.528,Z 424.027,A -85,B 0,C 180,E1 -12930.725,E2 -12930.725} C_VEL
LIN {X 0,Y 363.415,Z 417.176,A -85,B 0,C 180,E1 -12932.347,E2 -12932.347} C_VEL
LIN {X 0,Y 364.487,Z 408.64,A -85,B 0,C 180,E1 -12933.971,E2 -12933.971} C_VEL
LIN {X 0,Y 365.521,Z 399.181,A -85,B 0,C 180,E1 -12935.431,E2 -12935.431} C_VEL
LIN {X 0,Y 366.753,Z 388.593,A -85,B 0,C 180,E1 -12936.726,E2 -12936.726} C_VEL
LIN {X 0,Y 367.844,Z 377.275,A -85,B 0,C 180,E1 -12937.831,E2 -12937.831} C_VEL
LIN {X 0,Y 368.834,Z 364.794,A -85,B 0,C 180,E1 -12938.775,E2 -12938.775} C_VEL
LIN {X 0,Y 369.69,Z 350.827,A -85,B 0,C 180,E1 -12939.538,E2 -12939.538} C_VEL
LIN {X 0,Y 370.214,Z 338.07,A -85,B 0,C 180,E1 -12940.002,E2 -12940.002} C_VEL
LIN {X 0,Y 372.305,Z 255.199,A -85,B 0,C 180,E1 -12941.853,E2 -12941.853} C_VEL
LIN {X 0,Y 370.419,Z 247.473,A -85,B 0,C 180,E1 -12942.186,E2 -12942.186} C_VEL
LIN {X 0,Y 364.725,Z 234.05,A -85,B 0,C 180,E1 -12942.983,E2 -12942.983} C_VEL
LIN {X 0,Y 363.688,Z 231.568,A -85,B 0,C 180,E1 -12943.151,E2 -12943.151} C_VEL
LIN {X 0,Y 361.93,Z 224.407,A -85,B 0,C 180,E1 -12945.091,E2 -12945.091} C_VEL
LIN {X 0,Y 361.928,Z 224.409,A -85,B 0,C 180,E1 -12947.667,E2 -12947.667} C_VEL
LIN {X 0,Y 362.016,Z 224.396,A -85,B 0,C 180,E1 -12951.066,E2 -12951.066} C_VEL
LIN {X 0,Y 362.127,Z 224.378,A -85,B 0,C 180,E1 -12953.313,E2 -12953.313} C_VEL
LIN {X 0,Y 362.235,Z 224.364,A -85,B 0,C 180,E1 -12957.777,E2 -12957.777} C_VEL
LIN {X 0,Y 362.361,Z 224.348,A -85,B 0,C 180,E1 -12960,E2 -12960} C_VEL
LIN {X 0,Y 362.235,Z 224.364,A -85,B 0,C 180,E1 -12962.224,E2 -12962.224} C_VEL
